		;		
		// State Change Condition
		IF (me.Alarm.eActivAlmClass<>E_AlmClass.EOFF) AND (me.Alarm.eActivAlmClass<>E_AlmClass.OFF) THEN	
			IF(me.intCmd=cBCC_CMD_READ) THEN
				me.StateMachine.intStateNext := cBCC_STA_READBusy;
			END_IF
		END_IF
	END_IF

//--------------------------------------------------------------------------------------
// Exit action
	IF (me.StateMachine.intState<>me.StateMachine.intStateNext) THEN
		;
	END_IF
END_METHOD

METHOD PROTECTED sta_OFFBusy : BOOL
// state implemetation
//--------------------------------------------------------------------------------------
// Entry action
	IF (me.StateMachine.intState<>me.StateMachine.intStateLastCycle) THEN
		me.StateMachine.intStateLastCycle := me.StateMachine.intState;
		
		// Simulation timer	
		fbSimulationTimer.IN := FALSE;
		fbSimulationTimer.PT := UDINT_TO_TIME(SIf.Par.udiTORead_ms / 2);
		fbSimulationTimer(); // set time/reset timer
		fbSimulationTimer.IN := TRUE; // start timer
		
	END_IF

//--------------------------------------------------------------------------------------
// Cyclic action
	IF (me.StateMachine.intState=me.StateMachine.intStateLastCycle) THEN
		
		// Simulation
		IF (CIf.SwCfg.bolSimulation) THEN
			fbSimulationTimer(); // simulation time
			IF (fbSimulationTimer.Q) THEN
				pBCD_SIf^.intCmd := cBCD_CMD_DONE;
			END_IF
		END_IF
			
		// State Change Condition
		IF (pBCD_SIf^.stErr.bolErrorActive = TRUE) THEN
			me.StateMachine.intStateNext :=  cSTA_ERROR;
		ELSIF(pBCD_SIf^.intCmd = cBCD_CMD_DONE) THEN
			me.StateMachine.intStateNext := cSTA_OFF;
		END_IF
	END_IF

//--------------------------------------------------------------------------------------
// Exit action
	IF (me.StateMachine.intState<>me.StateMachine.intStateNext) THEN
		;
	END_IF
END_METHOD

METHOD PROTECTED sta_PON : BOOL
// state implemetation
//--------------------------------------------------------------------------------------
// Entry action
	IF (me.StateMachine.intState<>me.StateMachine.intStateLastCycle) THEN
		me.StateMachine.intStateLastCycle := me.StateMachine.intState;
		
	END_IF


//--------------------------------------------------------------------------------------
// Cyclic action
	IF (me.StateMachine.intState=me.StateMachine.intStateLastCycle) THEN
		
		;	
		// State Change Condition
		IF (me.intCmd<>cCMD_PON) AND (me.intCmd<>cCMD_DONE) THEN
			me.StateMachine.intStateNext := cSTA_OFFBusy;
		END_IF
	END_IF


//--------------------------------------------------------------------------------------
// Exit action
	IF (me.StateMachine.intState<>me.StateMachine.intStateNext) THEN
		;
	END_IF
END_METHOD

METHOD PROTECTED sta_PONBusy : BOOL
// state implemetation
//--------------------------------------------------------------------------------------
// Entry action
	IF (me.StateMachine.intState<>me.StateMachine.intStateLastCycle) THEN
		me.StateMachine.intStateLastCycle := me.StateMachine.intState;
		
		// Simulation timer	
		fbSimulationTimer.IN := FALSE;
		fbSimulationTimer.PT := UDINT_TO_TIME(SIf.Par.udiTORead_ms / 2);
		fbSimulationTimer(); // set time/reset timer
		fbSimulationTimer.IN := TRUE; // start timer
		
		// Reset driver status
		pBCD_SIf^.stStatus.bolSocketConnected := FALSE;
		pBCD_SIf^.stStatus.bolComChecked := FALSE;
	END_IF

//--------------------------------------------------------------------------------------
// Cyclic action
	IF (me.StateMachine.intState=me.StateMachine.intStateLastCycle) THEN
			
		// Simulation
		IF (CIf.SwCfg.bolSimulation) THEN
			fbSimulationTimer(); // simulation time
			IF (fbSimulationTimer.Q) THEN
				// Set driver status
				pBCD_SIf^.stStatus.bolSocketConnected := TRUE;
				pBCD_SIf^.stStatus.bolComChecked := TRUE;		
			END_IF
		END_IF
			
		// Try to open the TCP socket		
		pBCD_SIf^.intCmd := cBCD_CMD_CONNECT_SOCKET;  
					
		// Check if socket connected
		IF (pBCD_SIf^.stStatus.bolSocketConnected = TRUE) THEN
			pBCD_SIf^.intCmd :=	cBCD_CMD_COM_TEST; // Execute a communication test to see if the device answer		
		END_IF
		
		// State Change Condition
		IF ((pBCD_SIf^.stErr.bolErrorActive = TRUE) OR (me.StateMachine.udiTimeInState_ms >= SIf.Par.udiTOPowerOn_ms)) THEN
			// SIf.Alm[2].strText := 'Initialisation error from barcode reader. No answer from device.';
			pfbAlarmCtrl^.setAlarm(CIf.Info.intCtrlId,2,0,ADR(SIf.Alm),E_AlmState.RST,CIf.Job.eMe_ActivAlmClass);
			me.StateMachine.intStateNext := cSTA_ERROR;				
		ELSIF (pBCD_SIf^.stStatus.bolComChecked = TRUE) THEN
			me.StateMachine.intStateNext := cSTA_PON;
		END_IF
	END_IF

//--------------------------------------------------------------------------------------
// Exit action
	IF (me.StateMachine.intState<>me.StateMachine.intStateNext) THEN
		;
	END_IF
END_METHOD

METHOD PROTECTED sta_READ : BOOL
// state implemetation
//--------------------------------------------------------------------------------------
// Entry action
	IF (me.StateMachine.intState<>me.StateMachine.intStateLastCycle) THEN
		me.StateMachine.intStateLastCycle := me.StateMachine.intState;

	END_IF

//--------------------------------------------------------------------------------------
// Cyclic action
	IF (me.StateMachine.intState=me.StateMachine.intStateLastCycle) THEN

		// Simulation
		IF (CIf.SwCfg.bolSimulation) THEN
			;
		END_IF
		
		// State Change Condition
		IF(me.intCmd=cBCC_CMD_READ) THEN
			me.StateMachine.intStateNext := cBCC_STA_READBusy;
		END_IF
	END_IF

//--------------------------------------------------------------------------------------
// Exit action
	IF (me.StateMachine.intState<>me.StateMachine.intStateNext) THEN
		;
	END_IF
END_METHOD

METHOD PROTECTED sta_READBusy : BOOL
// state implemetation
//--------------------------------------------------------------------------------------
// Entry action
	IF (me.StateMachine.intState<>me.StateMachine.intStateLastCycle) THEN
		me.StateMachine.intStateLastCycle := me.StateMachine.intState;
		
		// Simulation timer	
		fbSimulationTimer.IN := FALSE;
		fbSimulationTimer.PT := UDINT_TO_TIME(SIf.Par.udiTORead_ms / 2);
		fbSimulationTimer(); // set time/reset timer
		fbSimulationTimer.IN := TRUE; // start timer
		
		// Init
		SIf.Cur.bolNewCodeReaded:= FALSE;
		SIf.Cur.bolNoRead:= FALSE;
		SIf.Cur.stData.uliBarCode:= 0;
		SIf.Cur.stData.strBarCode:= '';
		
		// Read barcode
		pBCD_SIf^.intCmd := cBCD_CMD_READ_BARCODE;
	END_IF


//--------------------------------------------------------------------------------------
// Cyclic action
	IF (me.StateMachine.intState=me.StateMachine.intStateLastCycle) THEN

		// Simulation
		IF (CIf.SwCfg.bolSimulation) THEN
			fbSimulationTimer(); // simulation time
			IF (fbSimulationTimer.Q) THEN
				SIf.Cur.bolNewCodeReaded:= TRUE;
				uliSimBarCode:= uliSimBarCode + 1;
				pBCD_SIf^.stData.uliBarCode:= uliSimBarCode;
				pBCD_SIf^.stData.strBarCode:= ULINT_TO_STRING(pBCD_SIf^.stData.uliBarCode);
				pBCD_SIf^.intCmd := cBCD_CMD_DONE;		
			END_IF
		END_IF	

		// Check for new barcode
		IF (pBCD_SIf^.stData.uliBarCode <> uliBarCodeOld) AND (pBCD_SIf^.stData.uliBarCode<>0) THEN
			uliBarCodeOld:= pBCD_SIf^.stData.uliBarCode;
			SIf.Cur.bolNewCodeReaded:= TRUE;
		END_IF
		
		// Get data from driver
		SIf.Cur.stData.uliBarCode:= pBCD_SIf^.stData.uliBarCode;
		SIf.Cur.stData.strBarCode:= pBCD_SIf^.stData.strBarCode;			
		
		// State Change Condition
		IF (pBCD_SIf^.stErr.bolErrorActive = TRUE) THEN  
			me.StateMachine.intStateNext :=  cSTA_ERROR;
		ELSIF (me.StateMachine.udiTimeInState_ms > SIf.Par.udiTORead_ms) THEN
			// SIf.Alm[4].strText := 'Timeout wait on data';
			pfbAlarmCtrl^.setAlarm(CIf.Info.intCtrlId,4,0,ADR(SIf.Alm),E_AlmState.RST,CIf.Job.eMe_ActivAlmClass);
			me.StateMachine.intStateNext :=  cSTA_ERROR;
		ELSIF (pBCD_SIf^.intCmd = cBCD_CMD_DONE) THEN
			IF (SIf.Cur.stData.uliBarCode=0) THEN
				SIf.Cur.bolNoRead:= TRUE;
				uliBarCodeOld:= 0;
				// SIf.Alm[3].strText := 'Barcode could not be read. Answer *NoRead* from device';
				pfbAlarmCtrl^.setAlarm(CIf.Info.intCtrlId,3,0,ADR(SIf.Alm),E_AlmState.RST,CIf.Job.eMe_ActivAlmClass);	
			END_IF		
			me.StateMachine.intStateNext := cBCC_STA_READ;
		END_IF
	END_IF

//--------------------------------------------------------------------------------------
// Exit action
	IF (me.StateMachine.intState<>me.StateMachine.intStateNext) THEN
		CIf.Job.intACmd:= cCMD_DONE;
		CIf.Job.intMCmd:= cCMD_DONE;
	END_IF
END_METHOD

METHOD PROTECTED StateMachine : BOOL
SUPER^.StateMachine();

// main statemachine of base controller
CASE me.StateMachine.intState OF
    cBCC_STA_READBusy: 
        THIS^.sta_READBusy();
    cBCC_STA_READ: 
        THIS^.sta_READ();	
END_CASE;
END_METHOD

END_FUNCTION_BLOCK

// POUs/Controller/Lvl0/CYL (Cylinder)/FB_CYL
FUNCTION_BLOCK FB_CYL EXTENDS FB_CtrlBase

VAR_INPUT
	In_bolRetracted: BOOL;
	In_bolExtended: BOOL;
END_VAR
VAR_OUTPUT
	Out_bolRetract: BOOL;
	Out_bolExtend: BOOL;
END_VAR

VAR
	/// Specific interface struct for public access
	SIf: T_Ctrl_SIf_CYL;
END_VAR

(*__________________________________________________________________________________________________
¦	
¦	Vistaprint Schweiz GmbH
¦	CH - 8401 Winterthur
¦
¦	www.vistaprint.ch - info@vistaprint.ch
¦___________________________________________________________________________________________________

Function desription:
Cylinder implementation. 


History:
Version		Date			Author		Comment
---------------------------------------------------------------------------------------------------
0.00.1		25.04.2013		AVME/KVO	Start history
0.00.2		03.07.2013		AVME/KVO	Always call Super.always, no change to off when switch to automatic
										alarm evt EOFF, OFF or cmd off detection in Always
0.00.3		05.11.2013		AVME/KVO	integrate in BaseElements library, 
										FB alarm pointer used, alarm definition over ENUM
___________________________________________________________________________________________________*)


IF (me.bolActivate) THEN // cyclic call enabled
	IF (CIf.Info.bolInitDone=FALSE) THEN // first cycle -> init
		CtrlInit();
		CIf.Info.bolInitDone := TRUE;
	ELSE
		CycleStartDuty();
	
		Always();
		
		StateMachine();
		
		CycleEndDuty();
	END_IF
END_IF;

METHOD PROTECTED Always : BOOL
IF (me.bolChangeBackToAUTO=TRUE) THEN // switch mode to automatic switch off controller
	//me.StateMachine.intStateNext := cSTA_OFFBusy;
	me.bolChangeBackToAUTO := FALSE; // for cylinder no change to off when switch to automatic!!
END_IF

SUPER^.Always();

// ----------------------------------------------------------------------------------
// cyclic actions outside of statemachine
IF (me.StateMachine.intState<>cSTA_SINGLE_ANSWER) THEN
	
	; // always error supervision
	
END_IF

// ----------------------------------------------------------------------------------
// overrule error always from base -> no EOFF State!! in EOFF go to OFF
IF (me.StateMachine.intStateNext = cSTA_EOFFBusy) THEN
	IF (me.StateMachine.intState=cSTA_OFF) THEN
		me.StateMachine.intStateNext := cSTA_OFF;
	ELSE // stay in OFF
		me.StateMachine.intStateNext := cSTA_OFFBusy;
	END_IF
END_IF
END_METHOD

METHOD FB_init : BOOL
VAR_INPUT
	///if TRUE, the retain variables are initialized (warm start / cold start)
	bInitRetains: BOOL;
	///if TRUE, the instance afterwards gets moved into the copy code (online change)
	bInCopyCode: BOOL;
END_VAR
VAR
	ii: UINT;
END_VAR
//------------------------------------------------------------------------------------------------------------------------
// to manually change in new FUB implementation!!!
// define valid commands for this controller
FOR ii:= 0 TO (SIZEOF(CIf.Job.aCmdList)/SIZEOF(CIf.Job.aCmdList[0])-1) BY 1 DO
	IF (CIf.Job.aCmdList[ii].intCmd=cCMD_INITIALIZED) THEN
		// found first empty array element
		EXIT;
	END_IF
END_FOR

CIf.Job.aCmdList[ii].intCmd := cCMD_STOP;
CIf.Job.aCmdList[ii].strName := 'Stop'; 
CIf.Job.aCmdList[ii].bolAvailable := TRUE;
ii := ii +1;
CIf.Job.aCmdList[ii].intCmd := cCMD_RETRACT;
CIf.Job.aCmdList[ii].strName := 'Retract';
CIf.Job.aCmdList[ii].bolAvailable := TRUE;
ii := ii +1;
CIf.Job.aCmdList[ii].intCmd := cCMD_EXTEND; // for test simulation single answer
CIf.Job.aCmdList[ii].strName := 'Extend';
CIf.Job.aCmdList[ii].bolAvailable := TRUE;

// set name of class/typ
CIf.Info.strType := 'FB_CYL'; 

// set alarm class
SIf.Alm[E_ALM_CYL.SensorRetractAlwaysOn].eAlmClass := E_AlmClass.TSTOP;
SIf.Alm[E_ALM_CYL.SensorRetractAlwaysOn].strText := 'sensor retract always on'; 
SIf.Alm[E_ALM_CYL.SensorExtendNotReached].eAlmClass := E_AlmClass.TSTOP;
SIf.Alm[E_ALM_CYL.SensorExtendNotReached].strText := 'timeout extend - sensor extend not reached';
SIf.Alm[E_ALM_CYL.SensorExtendAlwaysOn].eAlmClass := E_AlmClass.TSTOP;
SIf.Alm[E_ALM_CYL.SensorExtendAlwaysOn].strText := 'sensor extend always on';
SIf.Alm[E_ALM_CYL.SensorRetractNotReached].eAlmClass := E_AlmClass.TSTOP;
SIf.Alm[E_ALM_CYL.SensorRetractNotReached].strText := 'timeout retract - sensor retract not reached';
SIf.Alm[E_ALM_CYL.InterlockExtend].eAlmClass := E_AlmClass.OFF;
SIf.Alm[E_ALM_CYL.InterlockExtend].strText := 'interlock extend - movement stopped';
SIf.Alm[E_ALM_CYL.InterlockRetract].eAlmClass := E_AlmClass.OFF;
SIf.Alm[E_ALM_CYL.InterlockRetract].strText := 'interlock retract - movement stopped';

//*******************************************************************************
// initial values
//*******************************************************************************

// Configuration defaults of class
CIf.SwCfg.bolExist := TRUE;
CIf.SwCfg.bolEnable := TRUE;
CIf.SwCfg.bolSimulation := FALSE;

// Parameter defaults of class
SIf.Par.udiExtendTime_ms := 10000;
SIf.Par.udiRetractTime_ms := 8000;
SIf.Par.udiSimExtendTime_ms := SIf.Par.udiExtendTime_ms/2;	
SIf.Par.udiSimRetractTime_ms := SIf.Par.udiRetractTime_ms/2;
END_METHOD

METHOD PROTECTED getCmdState : STRING
VAR_INPUT
	intCmdState: INT;
	bolState: BOOL;
END_VAR
getCmdState := SUPER^.getCmdState(intCmdState:=intCmdState,bolState:=bolState); // get global/base defined cmds/states
IF (getCmdState='') THEN // global not defined get local
	// get string cmd/state string information in runtime
	IF (bolState=FALSE) THEN
		// cmd's
		CASE intCmdState OF
			CYL_CmdState.cCMD_RETRACT: 
				getCmdState := 'cCMD_RETRACT';
			CYL_CmdState.cCMD_EXTEND: 
				getCmdState := 'cCMD_EXTEND';
		ELSE
			getCmdState := 'Cmd not defined';
		END_CASE;
	ELSE
	
	// cmd's
		CASE intCmdState OF
			CYL_CmdState.cSTA_RETRACTBusy: 
				getCmdState := 'cSTA_RETRACTBusy';
			CYL_CmdState.cSTA_RETRACT: 
				getCmdState := 'cSTA_RETRACT';
			CYL_CmdState.cSTA_EXTENDBusy: 
				getCmdState := 'cSTA_EXTENDBusy';
			CYL_CmdState.cSTA_EXTEND: 
				getCmdState := 'cSTA_EXTEND';
		ELSE
			getCmdState := 'State not defined';
		END_CASE;
	END_IF
END_IF
END_METHOD

METHOD getCtrlSIf : POINTER TO T_Ctrl_SIf_CYL
getCtrlSIf := ADR(SIf);
END_METHOD

METHOD PROTECTED IoInBridge : BOOL
// digitale and analoge inputs read from hardware or forcing
SIf.In.bolExtended.map := THIS^.In_bolExtended;
SIf.In.bolRetracted.map := THIS^.In_bolRetracted;

IF (CIf.SwCfg.bolSimulation = FALSE) THEN
	getInBol(CIf.Job.bolIoForce,ADR(SIf.In.bolExtended));
	getInBol(CIf.Job.bolIoForce,ADR(SIf.In.bolRetracted));
ELSE
	//simulation of global IO
END_IF
END_METHOD

METHOD PROTECTED IoOutBridge : BOOL
VAR
	bolSwitchValvesOff: BOOL;
END_VAR
// digitale and analoge inputs read from hardware or forcing
IF (CIf.SwCfg.bolSimulation = FALSE) THEN
	setOutBol(CIf.Job.bolIoForce ,ADR(SIf.Out.bolExtend));
	setOutBol(CIf.Job.bolIoForce ,ADR(SIf.Out.bolRetract));
	
	// check interlocks to prevent damages
	IF (CIf.Job.bolIlkOverwrite=FALSE) THEN
		bolSwitchValvesOff := FALSE;
		
		IF (SIf.Ilk.bolExtend=TRUE) THEN
			// switch off?
			IF (SIf.Cfg.eTyp = E_Typ_CYL.Valve1_Sensor0) OR (SIf.Cfg.eTyp = E_Typ_CYL.Valve1_Sensor2) 
				OR (SIf.Cfg.eTyp = E_Typ_CYL.Valve1_SensorExtended) OR (SIf.Cfg.eTyp = E_Typ_CYL.Valve1_SensorRetracted) THEN
				// monostabil valve -> do nothing
			ELSE
				// bistable valve ->  switch both off
				bolSwitchValvesOff := TRUE;
				IF (SIf.Out.bolExtend.map=1) THEN
					pfbAlarmCtrl^.setAlarm(CIf.Info.intCtrlId,E_ALM_CYL.InterlockExtend,0,ADR(SIf.Alm),E_AlmState.RST,CIf.Job.eMe_ActivAlmClass);
				END_IF
			END_IF
		END_IF
		
		IF (SIf.Ilk.bolRetract=TRUE) THEN
			// switch off?
			IF (SIf.Cfg.eTyp = E_Typ_CYL.Valve1_Sensor0) OR (SIf.Cfg.eTyp = E_Typ_CYL.Valve1_Sensor2) 
				OR (SIf.Cfg.eTyp = E_Typ_CYL.Valve1_SensorExtended) OR (SIf.Cfg.eTyp = E_Typ_CYL.Valve1_SensorRetracted) THEN
				// monostabil valve -> do nothing
				;
			ELSE
				// bistable valve -> switch both off
				bolSwitchValvesOff := TRUE;
				IF (SIf.Out.bolRetract.map=1) THEN
					pfbAlarmCtrl^.setAlarm(CIf.Info.intCtrlId,E_ALM_CYL.InterlockRetract,0,ADR(SIf.Alm),E_AlmState.RST,CIf.Job.eMe_ActivAlmClass);
				END_IF;
			END_IF
		END_IF
		
		// bistable valve -> switch both off
		IF (bolSwitchValvesOff) THEN
			SIf.Out.bolExtend.map := FALSE;
			SIf.Out.bolRetract.map := FALSE;
		END_IF
		
	END_IF

	THIS^.Out_bolExtend := SIf.Out.bolExtend.map;
	THIS^.Out_bolRetract := SIf.Out.bolRetract.map;
END_IF
END_METHOD

METHOD PROTECTED sta_ERROR : BOOL
// state implemetation
//--------------------------------------------------------------------------------------
// Entry action
	IF (me.StateMachine.intState<>me.StateMachine.intStateLastCycle) THEN
		me.StateMachine.intStateHistory := me.StateMachine.intStateLastCycle; // -> possibillity to go back to state before error
		me.StateMachine.intStateLastCycle := me.StateMachine.intState;
		
	END_IF


//--------------------------------------------------------------------------------------
// Cyclic action
	IF (me.StateMachine.intState=me.StateMachine.intStateLastCycle) THEN
		
		;
		
		
		// State Change Condition
		IF (CIf.Job.bolAlmReset = TRUE) THEN
			me.StateMachine.intStateNext := cSTA_ERRORQuit;
		END_IF
	END_IF




//--------------------------------------------------------------------------------------
// Exit action
	IF (me.StateMachine.intState<>me.StateMachine.intStateNext) THEN
		;
	END_IF
END_METHOD

METHOD PROTECTED sta_ERRORQuit : BOOL
// state implemetation
//--------------------------------------------------------------------------------------
// Entry action
	IF (me.StateMachine.intState<>me.StateMachine.intStateLastCycle) THEN
		me.StateMachine.intStateLastCycle := me.StateMachine.intState;
		
	END_IF


//--------------------------------------------------------------------------------------
// Cyclic action
	IF (me.StateMachine.intState=me.StateMachine.intStateLastCycle) THEN
		
		;
		// evtl. wait time if reset of device is necessary and then decide to go to states or ERROR state
		IF (CIf.Job.bolAlmReset = TRUE) THEN
			CIf.Job.eMe_ActivAlmClass := E_AlmClass.NONE; // reset feedback channel for parent
			CIf.Job.bolAlmReset := FALSE;
		END_IF
		
		// State Change Condition
		IF (CIf.Job.bolAlmReset = FALSE) THEN
			IF (me.StateMachine.intStateHistory<=cSTA_PON) THEN
				me.StateMachine.intStateNext := cSTA_PONBusy;
			ELSIF(me.intCmd=cCMD_OFF) THEN
				me.StateMachine.intStateNext := cSTA_OFFBusy;
			ELSIF(me.intCmd=cCMD_STOP) THEN
				me.StateMachine.intStateNext := cSTA_STOPBusy;
			ELSIF(me.intCmd=cCMD_RETRACT) THEN
				me.StateMachine.intStateNext := cSTA_RETRACTBusy;
			ELSIF(me.intCmd=cCMD_EXTEND) THEN
				me.StateMachine.intStateNext := cSTA_EXTENDBusy;
			END_IF
		END_IF
	END_IF


//--------------------------------------------------------------------------------------
// Exit action
	IF (me.StateMachine.intState<>me.StateMachine.intStateNext) THEN
		;
	END_IF
END_METHOD

METHOD PROTECTED sta_EXTEND : BOOL
// state implemetation
//--------------------------------------------------------------------------------------
// Entry action
	IF (me.StateMachine.intState<>me.StateMachine.intStateLastCycle) THEN
		me.StateMachine.intStateLastCycle := me.StateMachine.intState;

	END_IF


//--------------------------------------------------------------------------------------
// Cyclic action
	IF (me.StateMachine.intState=me.StateMachine.intStateLastCycle) THEN

		// Simulation
		IF (CIf.SwCfg.bolSimulation) THEN
			;
		END_IF
		
		// State Change Condition
		IF (SIf.In.bolRetracted.intern) THEN
			// sensor retract always on
			pfbAlarmCtrl^.setAlarm(CIf.Info.intCtrlId,E_ALM_CYL.SensorRetractAlwaysOn,0,ADR(SIf.Alm),E_AlmState.RST,CIf.Job.eMe_ActivAlmClass);
			me.StateMachine.intStateNext :=  cSTA_ERROR;
		ELSIF ((SIf.In.bolExtended.intern = FALSE) AND ((SIf.Cfg.eTyp = E_Typ_CYL.Valve1_SensorExtended) OR (SIf.Cfg.eTyp = E_Typ_CYL.Valve2_SensorExtended))) THEN // wait time until error?
			me.StateMachine.intStateNext := CYL_CmdState.cSTA_EXTENDBusy;
		ELSIF(me.intCmd=cCMD_STOP) THEN
			me.StateMachine.intStateNext := cSTA_STOPBusy;
		ELSIF(me.intCmd=CYL_CmdState.cCMD_RETRACT) THEN
			me.StateMachine.intStateNext := CYL_CmdState.cSTA_RETRACTBusy;
		END_IF
	END_IF



//--------------------------------------------------------------------------------------
// Exit action
	IF (me.StateMachine.intState<>me.StateMachine.intStateNext) THEN
		;
	END_IF
END_METHOD

METHOD PROTECTED sta_EXTENDBusy : BOOL
// state implemetation
//--------------------------------------------------------------------------------------
// Entry action
	IF (me.StateMachine.intState<>me.StateMachine.intStateLastCycle) THEN
		me.StateMachine.intStateLastCycle := me.StateMachine.intState;

		fbSimulationTimer.IN := FALSE;
		fbSimulationTimer.PT := UDINT_TO_TIME(SIf.Par.udiSimExtendTime_ms);
		fbSimulationTimer(); // set time/reset timer
		fbSimulationTimer.IN := TRUE; // start timer
	END_IF


//--------------------------------------------------------------------------------------
// Cyclic action
	IF (me.StateMachine.intState=me.StateMachine.intStateLastCycle) THEN

		// Simulation
		IF (CIf.SwCfg.bolSimulation) THEN
			fbSimulationTimer(); // simulation time
			IF (fbSimulationTimer.Q) THEN
				SIf.In.bolExtended.intern := TRUE;
				SIf.In.bolRetracted.intern := FALSE;
			END_IF
		END_IF
		
		//no change action
		SIf.Out.bolExtend.intern := TRUE;
		SIf.Out.bolRetract.intern := FALSE;
		
		
		// State Change Condition
		IF (me.StateMachine.udiTimeInState_ms>SIf.Par.udiExtendTime_ms) THEN
			IF (SIf.In.bolRetracted.intern) THEN
				// sensor retract always on
				pfbAlarmCtrl^.setAlarm(CIf.Info.intCtrlId,E_ALM_CYL.SensorRetractAlwaysOn,0,ADR(SIf.Alm),E_AlmState.RST,CIf.Job.eMe_ActivAlmClass);
			ELSE
				// timeout extend
				pfbAlarmCtrl^.setAlarm(CIf.Info.intCtrlId,E_ALM_CYL.SensorExtendNotReached,0,ADR(SIf.Alm),E_AlmState.RST,CIf.Job.eMe_ActivAlmClass);
			END_IF
			me.StateMachine.intStateNext :=  cSTA_ERROR;
		ELSIF (SIf.In.bolExtended.intern) AND (SIf.In.bolRetracted.intern=FALSE) THEN
			me.StateMachine.intStateNext := CYL_CmdState.cSTA_EXTEND;
		ELSIF ((SIf.Cfg.eTyp = E_Typ_CYL.Valve1_SensorRetracted) OR (SIf.Cfg.eTyp = E_Typ_CYL.Valve2_SensorRetracted))
				 AND (SIf.In.bolRetracted.intern=FALSE) AND (me.StateMachine.udiTimeInState_ms>SIf.Par.udiSimExtendTime_ms) THEN
			me.StateMachine.intStateNext := CYL_CmdState.cSTA_EXTEND;
		ELSIF ((SIf.Cfg.eTyp = E_Typ_CYL.Valve1_Sensor0) OR (SIf.Cfg.eTyp = E_Typ_CYL.Valve2_Sensor0))
				AND (me.StateMachine.udiTimeInState_ms>SIf.Par.udiSimExtendTime_ms) THEN
			me.StateMachine.intStateNext := CYL_CmdState.cSTA_EXTEND;		
		ELSIF(me.intCmd=cCMD_STOP) THEN
			me.StateMachine.intStateNext := cSTA_STOPBusy;
		ELSIF(me.intCmd=cCMD_RETRACT) THEN
			me.StateMachine.intStateNext := CYL_CmdState.cSTA_RETRACTBusy;
		END_IF
	END_IF




//--------------------------------------------------------------------------------------
// Exit action
	IF (me.StateMachine.intState<>me.StateMachine.intStateNext) THEN
		SIf.Cur.udiMoveTimeExtend := me.StateMachine.udiTimeInState_ms;
	END_IF
END_METHOD

METHOD PROTECTED sta_OFF : BOOL
// state implemetation
//--------------------------------------------------------------------------------------
// Entry action
	IF (me.StateMachine.intState<>me.StateMachine.intStateLastCycle) THEN
		me.StateMachine.intStateLastCycle := me.StateMachine.intState;
		
	END_IF


//--------------------------------------------------------------------------------------
// Cyclic action
	IF (me.StateMachine.intState=me.StateMachine.intStateLastCycle) THEN
		
		;
		
		// State Change Condition
		IF (me.Alarm.eActivAlmClass<>E_AlmClass.EOFF) AND (me.Alarm.eActivAlmClass<>E_AlmClass.OFF) THEN
			IF (me.intCmd=cCMD_STOP) THEN
				// sensor retract always on cylinder
				me.StateMachine.intStateNext :=  cSTA_STOPBusy;
			ELSIF (me.intCmd=CYL_CmdState.cCMD_EXTEND) THEN 
				me.StateMachine.intStateNext := cSTA_EXTENDBusy;
			ELSIF(me.intCmd=CYL_CmdState.cCMD_RETRACT) THEN
				me.StateMachine.intStateNext := cSTA_RETRACTBusy;
			END_IF
		END_IF
	END_IF




//--------------------------------------------------------------------------------------
// Exit action
	IF (me.StateMachine.intState<>me.StateMachine.intStateNext) THEN
		;
	END_IF
END_METHOD

METHOD PROTECTED sta_OFFBusy : BOOL
// state implemetation
//--------------------------------------------------------------------------------------
// Entry action
	IF (me.StateMachine.intState<>me.StateMachine.intStateLastCycle) THEN
		me.StateMachine.intStateLastCycle := me.StateMachine.intState;
		
	END_IF


//--------------------------------------------------------------------------------------
// Cyclic action
	IF (me.StateMachine.intState=me.StateMachine.intStateLastCycle) THEN
		
		// switch off?
		IF (SIf.Cfg.eTyp = E_Typ_CYL.Valve1_Sensor0) OR (SIf.Cfg.eTyp = E_Typ_CYL.Valve1_Sensor2) 
			OR (SIf.Cfg.eTyp = E_Typ_CYL.Valve1_SensorExtended) OR (SIf.Cfg.eTyp = E_Typ_CYL.Valve1_SensorRetracted) THEN
			// monostabil valve -> do nothing
			;
		ELSE
			// bistable valve -> switch both off
			SIf.Out.bolExtend.intern := FALSE;
			SIf.Out.bolRetract.intern := FALSE;
		END_IF
		
		
		
		// State Change Condition
		IF (TRUE) THEN
			me.StateMachine.intStateNext := cSTA_OFF;
		END_IF
	END_IF




//--------------------------------------------------------------------------------------
// Exit action
	IF (me.StateMachine.intState<>me.StateMachine.intStateNext) THEN
		;
	END_IF
END_METHOD

METHOD PROTECTED sta_PON : BOOL
// state implemetation
//--------------------------------------------------------------------------------------
// Entry action
	IF (me.StateMachine.intState<>me.StateMachine.intStateLastCycle) THEN
		me.StateMachine.intStateLastCycle := me.StateMachine.intState;
		
	END_IF


//--------------------------------------------------------------------------------------
// Cyclic action
	IF (me.StateMachine.intState=me.StateMachine.intStateLastCycle) THEN
		
		;
		
		// State Change Condition
		IF(me.intCmd=cCMD_STOP) THEN
			me.StateMachine.intStateNext := cSTA_STOPBusy;
		ELSIF(me.intCmd=cCMD_RETRACT) THEN
			me.StateMachine.intStateNext := cSTA_RETRACTBusy;
		ELSIF (me.intCmd=cCMD_EXTEND) THEN
			me.StateMachine.intStateNext := cSTA_EXTENDBusy;
		END_IF
	END_IF




//--------------------------------------------------------------------------------------
// Exit action
	IF (me.StateMachine.intState<>me.StateMachine.intStateNext) THEN
		;
	END_IF
END_METHOD

METHOD PROTECTED sta_RETRACT : BOOL
// state implemetation
//--------------------------------------------------------------------------------------
// Entry action
	IF (me.StateMachine.intState<>me.StateMachine.intStateLastCycle) THEN
		me.StateMachine.intStateLastCycle := me.StateMachine.intState;

	END_IF


//--------------------------------------------------------------------------------------
// Cyclic action
	IF (me.StateMachine.intState=me.StateMachine.intStateLastCycle) THEN

		// Simulation
		IF (CIf.SwCfg.bolSimulation) THEN
			;
		END_IF
		
		// State Change Condition
		IF (SIf.In.bolExtended.intern) THEN
			// sensor retract always on
			pfbAlarmCtrl^.setAlarm(CIf.Info.intCtrlId,E_ALM_CYL.SensorExtendAlwaysOn,0,ADR(SIf.Alm),E_AlmState.RST,CIf.Job.eMe_ActivAlmClass);
			me.StateMachine.intStateNext :=  cSTA_ERROR;
		ELSIF ((SIf.In.bolRetracted.intern = FALSE) AND ((SIf.Cfg.eTyp = E_Typ_CYL.Valve1_SensorRetracted) OR (SIf.Cfg.eTyp = E_Typ_CYL.Valve2_SensorRetracted))) THEN // wait time until error?
			me.StateMachine.intStateNext := CYL_CmdState.cSTA_RETRACTBusy;
		ELSIF(me.intCmd=cCMD_STOP) THEN
			me.StateMachine.intStateNext := cSTA_STOPBusy;
		ELSIF(me.intCmd=CYL_CmdState.cCMD_EXTEND) THEN
			me.StateMachine.intStateNext := CYL_CmdState.cSTA_EXTENDBusy;
		END_IF
	END_IF




//--------------------------------------------------------------------------------------
// Exit action
	IF (me.StateMachine.intState<>me.StateMachine.intStateNext) THEN
		;
	END_IF
END_METHOD

METHOD PROTECTED sta_RETRACTBusy : BOOL
// state implemetation
//--------------------------------------------------------------------------------------
// Entry action
	IF (me.StateMachine.intState<>me.StateMachine.intStateLastCycle) THEN
		me.StateMachine.intStateLastCycle := me.StateMachine.intState;
		
		SIf.Out.bolExtend.intern := FALSE;
		SIf.Out.bolRetract.intern := TRUE;
		
		fbSimulationTimer.IN := FALSE;
		fbSimulationTimer.PT := UDINT_TO_TIME(SIf.Par.udiSimRetractTime_ms);
		fbSimulationTimer(); // set time/reset timer
		fbSimulationTimer.IN := TRUE; // start timer
	END_IF


//--------------------------------------------------------------------------------------
// Cyclic action
	IF (me.StateMachine.intState=me.StateMachine.intStateLastCycle) THEN

		// Simulation
		IF (CIf.SwCfg.bolSimulation) THEN
			fbSimulationTimer(); // simulation time
			IF (fbSimulationTimer.Q) THEN
				SIf.In.bolRetracted.intern := TRUE;
				SIf.In.bolExtended.intern := FALSE;
			END_IF
		END_IF
		
		// State Change Condition
		IF (me.StateMachine.udiTimeInState_ms>SIf.Par.udiRetractTime_ms) THEN
			IF (SIf.In.bolExtended.intern) THEN
				// sensor extend always on 
				pfbAlarmCtrl^.setAlarm(CIf.Info.intCtrlId,E_ALM_CYL.SensorExtendAlwaysOn,0,ADR(SIf.Alm),E_AlmState.RST,CIf.Job.eMe_ActivAlmClass);
			ELSE
				// timeout retract cylinder
				pfbAlarmCtrl^.setAlarm(CIf.Info.intCtrlId,E_ALM_CYL.SensorRetractNotReached,0,ADR(SIf.Alm),E_AlmState.RST,CIf.Job.eMe_ActivAlmClass);
			END_IF
			me.StateMachine.intStateNext :=  cSTA_ERROR;
		ELSIF (SIf.In.bolRetracted.intern) AND(SIf.In.bolExtended.intern=FALSE) THEN
			me.StateMachine.intStateNext := CYL_CmdState.cSTA_RETRACT;
		ELSIF ((SIf.Cfg.eTyp = E_Typ_CYL.Valve1_SensorExtended) OR (SIf.Cfg.eTyp = E_Typ_CYL.Valve2_SensorExtended))
				 AND (SIf.In.bolExtended.intern=FALSE) AND (me.StateMachine.udiTimeInState_ms>SIf.Par.udiSimRetractTime_ms) THEN
			me.StateMachine.intStateNext := CYL_CmdState.cSTA_RETRACT;
		ELSIF ((SIf.Cfg.eTyp = E_Typ_CYL.Valve1_Sensor0) OR (SIf.Cfg.eTyp = E_Typ_CYL.Valve2_Sensor0))
				AND (me.StateMachine.udiTimeInState_ms>SIf.Par.udiSimRetractTime_ms) THEN
			me.StateMachine.intStateNext := CYL_CmdState.cSTA_RETRACT;		
		ELSIF(me.intCmd=cCMD_STOP) THEN
			me.StateMachine.intStateNext := cSTA_STOPBusy;
		ELSIF(me.intCmd=CYL_CmdState.cCMD_EXTEND) THEN
			me.StateMachine.intStateNext := CYL_CmdState.cSTA_EXTENDBusy;
		END_IF
	END_IF




//--------------------------------------------------------------------------------------
// Exit action
	IF (me.StateMachine.intState<>me.StateMachine.intStateNext) THEN
		SIf.Cur.udiMoveTimeRetract := me.StateMachine.udiTimeInState_ms;
	END_IF
END_METHOD

METHOD PROTECTED sta_STOP : BOOL
// state implemetation
//--------------------------------------------------------------------------------------
// Entry action
	IF (me.StateMachine.intState<>me.StateMachine.intStateLastCycle) THEN
		me.StateMachine.intStateLastCycle := me.StateMachine.intState;
		
	END_IF


//--------------------------------------------------------------------------------------
// Cyclic action
	IF (me.StateMachine.intState=me.StateMachine.intStateLastCycle) THEN
		
		;
		
		
		// State Change Condition
		IF (me.intCmd=CYL_CmdState.cCMD_EXTEND) THEN 
			me.StateMachine.intStateNext := CYL_CmdState.cSTA_EXTENDBusy;
		ELSIF(me.intCmd=CYL_CmdState.cCMD_RETRACT) THEN
			me.StateMachine.intStateNext := CYL_CmdState.cSTA_RETRACTBusy;
		END_IF
	END_IF




//--------------------------------------------------------------------------------------
// Exit action
	IF (me.StateMachine.intState<>me.StateMachine.intStateNext) THEN
		;
	END_IF
END_METHOD

METHOD PROTECTED sta_STOPBusy : BOOL
// state implemetation
//--------------------------------------------------------------------------------------
// Entry action
	IF (me.StateMachine.intState<>me.StateMachine.intStateLastCycle) THEN
		me.StateMachine.intStateLastCycle := me.StateMachine.intState;
		
	END_IF


//--------------------------------------------------------------------------------------
// Cyclic action
	IF (me.StateMachine.intState=me.StateMachine.intStateLastCycle) THEN
		
		// switch off?
		IF (SIf.Cfg.eTyp = E_Typ_CYL.Valve1_Sensor0) OR (SIf.Cfg.eTyp = E_Typ_CYL.Valve1_Sensor2) 
			OR (SIf.Cfg.eTyp = E_Typ_CYL.Valve1_SensorExtended) OR (SIf.Cfg.eTyp = E_Typ_CYL.Valve1_SensorRetracted) THEN
			// monostabil valve -> do nothing
			;
		ELSE
			// bistable valve -> switch both on -> block at position
			SIf.Out.bolExtend.intern := TRUE;
			SIf.Out.bolRetract.intern := TRUE;
		END_IF
		
		
		
		// State Change Condition
		IF (TRUE) THEN
			me.StateMachine.intStateNext := cSTA_STOP;
		END_IF
	END_IF




//--------------------------------------------------------------------------------------
// Exit action
	IF (me.StateMachine.intState<>me.StateMachine.intStateNext) THEN
		;
	END_IF
END_METHOD

METHOD PROTECTED StateMachine : BOOL
SUPER^.StateMachine();

// main statemachine of base controller
CASE me.StateMachine.intState OF
    CYL_CmdState.cSTA_RETRACTBusy: 
        THIS^.sta_RETRACTBusy();
    CYL_CmdState.cSTA_RETRACT: 
        THIS^.sta_RETRACT();
    CYL_CmdState.cSTA_EXTENDBusy: 
        THIS^.sta_EXTENDBusy();
    CYL_CmdState.cSTA_EXTEND: 
        THIS^.sta_EXTEND();
	cSTA_STOPBusy: 
        THIS^.sta_STOPBusy();
    cSTA_STOP: 
        THIS^.sta_STOP();
END_CASE;
END_METHOD

END_FUNCTION_BLOCK

// POUs/Controller/Lvl0/DRV (Drive)/FB_DRV
FUNCTION_BLOCK FB_DRV EXTENDS FB_CtrlBase
VAR_INPUT
	In_bolOverload: BOOL;
	In_bolPulse: BOOL;
	In_a_bolBlockedSupvervis: ARRAY[1..cMAX_BLOCKED_SUP] OF BOOL;
END_VAR
VAR_OUTPUT
	Out_bolSpeed_1: BOOL;
	Out_bolSpeed_2: BOOL;
END_VAR
VAR
	/// Specific interface struct for public access
	SIf: T_Ctrl_SIf_DRV;
	bolPulseFlag: BOOL;
	udiPulseTimeoutTimer: UDINT;
	/// Timer for speed average calculation
	udiTimerSpeedCalc: UDINT;
	/// Shift register for average calculation of the speed
	aSpeedShift: ARRAY[0..4] OF DINT;
	/// Size of Speed Shift array for average calculation
	intSpeedShiftSize: INT;
	/// Varible for Speedcalculation
	dinSpeedCalc_um_s: DINT;
	/// Varible for Speedcalculation
	dinSpeedNew_um_s: DINT;
	/// Old Position for Speed calculation
	dinPosOld_um: DINT;
	/// Loop variable
	intI: INT;
	/// Blocked supervision
	/// Array with supervision distances
	a_dintPinDistance: ARRAY[1..cMAX_BLOCKED_SUP] OF DINT;
	a_bolREBlockedSupvervis: ARRAY[1..cMAX_BLOCKED_SUP] OF BOOL;
	/// Old Position for from last cycle
	dinPosOldCycle_um: DINT;
END_VAR
VAR CONSTANT
	/// Check speed every 250ms
	cSpeedCalcTime_ms: UDINT := 250;
END_VAR

(*__________________________________________________________________________________________________
¦	
¦	Vistaprint Schweiz GmbH
¦	CH - 8401 Winterthur
¦
¦	www.vistaprint.ch - info@vistaprint.ch
¦___________________________________________________________________________________________________

Function desription:
Drive element for all different Drive types, 
Configuration of the type and Speed Calculation


History:
Version		Date			Author		Comment
---------------------------------------------------------------------------------------------------
0.00.1		27.06.2013		VP/RE		Start history
0.00.2		28.08.2013		AVME/PRE	Implement speed calculation
0.00.3		19.09.2013		AVME/PRE	Implement new Base Concept
0.00.4		02.10.2013		VP/RE		Added pulse counter. Changed pulse distance to 28.4 mm as a default value. Changed driving distance to 305 mm.
0.00.5      10.10.2013		AVME/DSC    In_bolBufferFull deleted. Not needed in DRV controller. Handled by parent controller if necessary.
0.00.6      18.10.2013		AVME/DSC    SIf.Alm[4].strText deleted in FB_init. Not used anymore.
0.00.7		22.10.2013		AVME/MRU	DRV without pulse sensor simulated pulse imroved
0.00.8      23.10.2013		AVME/DSC    Speed calculation from always to state RUN. cSpeedCalcTime_ms -> 250ms. Shift register array 0..4. Clear buffer in state RUN entry action.
										Changes for better position interpolation in controllers like MER, DPJ, DHC and JUN.
___________________________________________________________________________________________________*)


IF (me.bolActivate) THEN // cyclic call enabled
	IF (CIf.Info.bolInitDone=FALSE) THEN // first cycle -> init
		CtrlInit();
		CIf.Info.bolInitDone := TRUE;
	ELSE
		CycleStartDuty();
	
		Always();
		
		StateMachine();
		
		CycleEndDuty();
	END_IF
END_IF;

METHOD PROTECTED Always : BOOL
SUPER^.Always();

IF (me.StateMachine.intState<>cSTA_SINGLE_ANSWER) THEN
	
	// Error checks not in OFF and Error States
	IF (me.StateMachine.intState<>cSTA_OFF) AND (me.StateMachine.intState<>cSTA_ERROR) AND (me.StateMachine.intState<>cSTA_ERRORQuit) THEN
		IF SIf.In.bolOverload.intern THEN
			// SIf.Alm[1].strText := 'Drive overload'; 
			pfbAlarmCtrl^.setAlarm(CIf.Info.intCtrlId,1,0,ADR(SIf.Alm),E_AlmState.RST,CIf.Job.eMe_ActivAlmClass);		
			me.StateMachine.intStateNext := cSTA_ERROR;		
		END_IF
		
		// Blocked Supervision control
		// Sensor detect Pins, if a defined count of pins are brocken, the machine stops
		FOR intI := 1 TO SIf.Cfg.usiCountBlockedSupervis DO
			
			// Simulation
			// Simulate the Pins in the drive
			IF (CIf.SwCfg.bolSimulation) THEN
				IF (a_dintPinDistance[intI] >  SIf.Cfg.dinPinDistance_um) THEN
					SIf.In.a_bolBlockedSupvervis[intI].intern := TRUE;
				ELSE
					SIf.In.a_bolBlockedSupvervis[intI].intern := FALSE;
				END_IF
			END_IF
		
			// Check if a new pin is arrive, set distance to last pin to '0'
			IF ((SIf.In.a_bolBlockedSupvervis[intI].intern = TRUE) AND (a_bolREBlockedSupvervis[intI] = FALSE)) THEN
				a_bolREBlockedSupvervis[intI] := TRUE;
				a_dintPinDistance[intI] := 0;
			ELSIF ((SIf.In.a_bolBlockedSupvervis[intI].intern = FALSE) AND (a_bolREBlockedSupvervis[intI] = TRUE)) THEN
				a_bolREBlockedSupvervis[intI] := FALSE;
			END_IF
			// Check distance to last Pin, if to far away, set error
			IF (a_dintPinDistance[intI] > ((SIf.Par.int_MaxBrokenPins+1) * SIf.Cfg.dinPinDistance_um)) THEN
				// SIf.Alm[3].strText := 'Drive blocked, Pins are broken'; 
				pfbAlarmCtrl^.setAlarm(CIf.Info.intCtrlId,3,0,ADR(SIf.Alm),E_AlmState.RST,CIf.Job.eMe_ActivAlmClass);
				a_dintPinDistance[intI] := 0;		
				me.StateMachine.intStateNext := cSTA_ERROR;		
			ELSE
				a_dintPinDistance[intI] := a_dintPinDistance[intI] + SIf.Cur.dinPos_um - dinPosOldCycle_um;					
			END_IF		
		END_FOR
		dinPosOldCycle_um := SIf.Cur.dinPos_um;
	END_IF
END_IF

// Speed calculation in always function to get correct position everytime, not only in run
// observe no pulse detected failure case 
IF (SIf.In.bolPulse.intern AND NOT(bolPulseFlag)) THEN				
	// calculate CUR
	SIf.Cur.dinPos_um := SIf.Cur.dinPos_um + SIf.Cfg.dinDistPerPulse_um;
	SIf.Cur.dinPulseCounter := SIf.Cur.dinPulseCounter + 1;
		
	udiPulseTimeoutTimer := 0;
	bolPulseFlag := TRUE;
ELSIF (NOT(SIf.In.bolPulse.intern) AND bolPulseFlag) THEN
	bolPulseFlag := FALSE;
END_IF

// Always change actions in Base Library
// ----------------------------------------------------------------------------------
// overrule error always from base -> no EOFF State!! in EOFF go to OFF
IF (me.StateMachine.intStateNext = cSTA_EOFFBusy) THEN
	IF (me.StateMachine.intState=cSTA_OFF) THEN
		me.StateMachine.intStateNext := cSTA_OFF;
	ELSE // stay in OFF
		me.StateMachine.intStateNext := cSTA_OFFBusy;
	END_IF
END_IF
END_METHOD

METHOD FB_init : BOOL
VAR_INPUT
	///if TRUE, the retain variables are initialized (warm start / cold start)
	bInitRetains: BOOL;
	///if TRUE, the instance afterwards gets moved into the copy code (online change)
	bInCopyCode: BOOL;
END_VAR
VAR
	ii: UINT;
END_VAR
//------------------------------------------------------------------------------------------------------------------------
// to manually change in new FUB implementation!!!
// define valid commands for this controller
FOR ii:= 0 TO (SIZEOF(CIf.Job.aCmdList)/SIZEOF(CIf.Job.aCmdList[0])-1) BY 1 DO
	IF (CIf.Job.aCmdList[ii].intCmd=cCMD_INITIALIZED) THEN
		// found first empty array element
		EXIT;
	END_IF
END_FOR
CIf.Job.aCmdList[ii].intCmd := cCMD_RUN;
CIf.Job.aCmdList[ii].strName := 'Run'; 
CIf.Job.aCmdList[ii].bolAvailable := TRUE;
ii := ii +1;

// set name of class/typ
CIf.Info.strType := 'FB_DRV'; 

// set alarm class
SIf.Alm[1].eAlmClass := E_AlmClass.OFF;
SIf.Alm[1].strText := 'Drive overload'; 
SIf.Alm[2].eAlmClass := E_AlmClass.OFF;
SIf.Alm[2].strText := 'Timeout no pulse detected';
SIf.Alm[3].eAlmClass := E_AlmClass.OFF;
SIf.Alm[3].strText := 'Drive blocked, Pins are broken'; 

//*******************************************************************************
// initial values
//*******************************************************************************

// software configuration
CIf.SwCfg.bolExist := TRUE;
CIf.SwCfg.bolSimulation := FALSE;

// parmeter
SIf.Par.udi_pulseTimeout_ms := 2000;
SIf.Par.udi_pulseSim_ms := 56;
SIf.Par.usi_speedLevel := 0;
SIf.Par.int_MaxBrokenPins := 5;

SIf.Cfg.dinDistPerPulse_um := 28400; // 28,4[mm/puls]
SIf.Cfg.usiCountBlockedSupervis := 0;
SIf.Cfg.dinPinDistance_um := 305000;
END_METHOD

METHOD getCtrlSIf : POINTER TO T_Ctrl_SIf_DRV
getCtrlSIf := ADR(SIf);
END_METHOD

METHOD PROTECTED IoInBridge : BOOL
// digitale and analoge inputs read from hardware or forcing
SIf.In.bolOverload.map := THIS^.In_bolOverload;
SIf.In.bolPulse.map := THIS^.In_bolPulse;

FOR intI := 1 TO SIf.Cfg.usiCountBlockedSupervis DO
	SIf.In.a_bolBlockedSupvervis[intI].map := THIS^.In_a_bolBlockedSupvervis[intI];
	IF (CIf.SwCfg.bolSimulation = FALSE) THEN
		getInBol(CIf.Job.bolIoForce,ADR(SIf.In.a_bolBlockedSupvervis[intI]));
	END_IF
END_FOR

IF (CIf.SwCfg.bolSimulation = FALSE) THEN
	getInBol(CIf.Job.bolIoForce,ADR(SIf.In.bolOverload));
	getInBol(CIf.Job.bolIoForce,ADR(SIf.In.bolPulse));
	//ctrl.In.bol_PosSwitchBasicDefTyp.intern := getInBol(ctrl.ifc.Job.bol_Force ,ADR(ctrl.In.bol_PosSwitchBasicDefTyp);
ELSE
	//simulation of global IO
	SIf.In.bolOverload.intern := FALSE;
END_IF
END_METHOD

METHOD PROTECTED IoOutBridge : BOOL
VAR
	bolSwitchValvesOff: BOOL;
END_VAR
// digitale and analoge inputs read from hardware or forcing
IF (CIf.SwCfg.bolSimulation = FALSE) THEN
	setOutBol(CIf.Job.bolIoForce ,ADR(SIf.Out.bolSpeed_1));
	setOutBol(CIf.Job.bolIoForce ,ADR(SIf.Out.bolSpeed_2));

	THIS^.Out_bolSpeed_1 := SIf.Out.bolSpeed_1.map;
	THIS^.Out_bolSpeed_2 := SIf.Out.bolSpeed_2.map;
END_IF
END_METHOD

METHOD PRIVATE SetSpeed
// 0=slow, 1=middle, 2=fast
CASE SIf.Par.usi_speedLevel OF
	0:
		SIf.Out.bolSpeed_1.intern := TRUE;
		SIf.Out.bolSpeed_2.intern := FALSE;
	1:
		SIf.Out.bolSpeed_1.intern := TRUE;
		SIf.Out.bolSpeed_2.intern := TRUE;
	2:
		SIf.Out.bolSpeed_1.intern := FALSE;
		SIf.Out.bolSpeed_2.intern := TRUE;
	ELSE
		SIf.Out.bolSpeed_1.intern := TRUE;
		SIf.Out.bolSpeed_2.intern := FALSE;
END_CASE
END_METHOD

METHOD PROTECTED sta_ERROR : BOOL
// state implemetation
//--------------------------------------------------------------------------------------
// Entry action
IF (me.StateMachine.intState<>me.StateMachine.intStateLastCycle) THEN
	me.StateMachine.intStateHistory := me.StateMachine.intStateLastCycle; // -> possibillity to go back to state before error
	me.StateMachine.intStateLastCycle := me.StateMachine.intState;
	
	SIf.Out.bolSpeed_1.intern := FALSE;
	SIf.Out.bolSpeed_2.intern := FALSE;
	
END_IF


//--------------------------------------------------------------------------------------
// Cyclic action
	IF (me.StateMachine.intState=me.StateMachine.intStateLastCycle) THEN
		
		;
		
		
		// State Change Condition
		IF (CIf.Job.bolAlmReset = TRUE) THEN
			me.StateMachine.intStateNext := cSTA_ERRORQuit;
		END_IF
	END_IF




//--------------------------------------------------------------------------------------
// Exit action
	IF (me.StateMachine.intState<>me.StateMachine.intStateNext) THEN
		;
	END_IF
END_METHOD

METHOD PROTECTED sta_OFF : BOOL
// state implemetation
//--------------------------------------------------------------------------------------
// Entry action
	IF (me.StateMachine.intState<>me.StateMachine.intStateLastCycle) THEN
		me.StateMachine.intStateLastCycle := me.StateMachine.intState;
		
	END_IF


//--------------------------------------------------------------------------------------
// Cyclic action
	IF (me.StateMachine.intState=me.StateMachine.intStateLastCycle) THEN
		
		;
		
		
		// State Change Condition
		IF (me.Alarm.eActivAlmClass<>E_AlmClass.EOFF) AND (me.Alarm.eActivAlmClass<>E_AlmClass.OFF) THEN
			IF (me.intCmd=cCMD_RUN) THEN 
				me.StateMachine.intStateNext := cSTA_RUNBusy;
			END_IF
		END_IF
	END_IF




//--------------------------------------------------------------------------------------
// Exit action
	IF (me.StateMachine.intState<>me.StateMachine.intStateNext) THEN
		;
	END_IF
END_METHOD

METHOD PROTECTED sta_OFFBusy : BOOL
// state implemetation
//--------------------------------------------------------------------------------------
// Entry action
	IF (me.StateMachine.intState<>me.StateMachine.intStateLastCycle) THEN
		me.StateMachine.intStateLastCycle := me.StateMachine.intState;
		
	END_IF


//--------------------------------------------------------------------------------------
// Cyclic action
	IF (me.StateMachine.intState=me.StateMachine.intStateLastCycle) THEN
		
		SIf.Out.bolSpeed_1.intern := FALSE;
		SIf.Out.bolSpeed_2.intern := FALSE;
		
		// State Change Condition
		IF (TRUE) THEN
			me.StateMachine.intStateNext := cSTA_OFF;
		END_IF
	END_IF




//--------------------------------------------------------------------------------------
// Exit action
	IF (me.StateMachine.intState<>me.StateMachine.intStateNext) THEN
		;
	END_IF
END_METHOD

METHOD PROTECTED sta_PON : BOOL
// state implemetation
//--------------------------------------------------------------------------------------
// Entry action
	IF (me.StateMachine.intState<>me.StateMachine.intStateLastCycle) THEN
		me.StateMachine.intStateLastCycle := me.StateMachine.intState;
		
	END_IF


//--------------------------------------------------------------------------------------
// Cyclic action
	IF (me.StateMachine.intState=me.StateMachine.intStateLastCycle) THEN
		
		;
		
		
		// State Change Condition
		IF ((me.intCmd=cCMD_OFF) OR (me.intCmd=cCMD_RUN)) THEN
			me.StateMachine.intStateNext := cSTA_OFFBusy;
		END_IF
	END_IF




//--------------------------------------------------------------------------------------
// Exit action
	IF (me.StateMachine.intState<>me.StateMachine.intStateNext) THEN
		;
	END_IF
END_METHOD

METHOD PROTECTED sta_RUN : BOOL
VAR
	ii: INT;
END_VAR
// state implemetation
//--------------------------------------------------------------------------------------
// Entry action
	IF (me.StateMachine.intState<>me.StateMachine.intStateLastCycle) THEN
		me.StateMachine.intStateLastCycle := me.StateMachine.intState;
		
		udiPulseTimeoutTimer := 0;
		bolPulseFlag := FALSE;
		
		fbSimulationTimer.IN := FALSE;
		fbSimulationTimer.PT := UDINT_TO_TIME(SIf.Par.udi_pulseSim_ms);  
		fbSimulationTimer(); // set time/reset timer
		fbSimulationTimer.IN := TRUE; // start timer
			
		// Get Size of array
		intSpeedShiftSize := SIZEOF(aSpeedShift)/(SIZEOF(aSpeedShift[0]));
		// Clear speed buffer
		FOR ii:=0 TO intSpeedShiftSize-1 BY 1 DO
			aSpeedShift[ii]:=0;
		END_FOR
		
	END_IF


//--------------------------------------------------------------------------------------
// Cyclic action
	IF (me.StateMachine.intState=me.StateMachine.intStateLastCycle) THEN
		
		// Simulation
		// AND speed simulation if no distance sensor is existing !!!
		IF ((CIf.SwCfg.bolSimulation) OR (SIf.Cfg.bolPulseExist = FALSE)) THEN
			fbSimulationTimer(); // simulation time
			IF (fbSimulationTimer.Q) THEN
				SIf.In.bolPulse.intern := TRUE; 
				In_bolPulse := TRUE; // MRU 22.10.2013 added for drive without pulse sensor
				fbSimulationTimer.IN := FALSE;
			ELSE
				SIf.In.bolPulse.intern := FALSE;
				In_bolPulse := FALSE; // MRU 22.10.2013 added for drive without pulse sensor
				fbSimulationTimer.IN := TRUE;
			END_IF
		END_IF
	
		IF SIf.Cfg.bolSpeedVariable = TRUE THEN
			SetSpeed();
		END_IF;
		
		udiPulseTimeoutTimer := udiPulseTimeoutTimer + me.FUBInfo.udiSample_ms;
		
		
		// Speed calculation
		IF udiTimerSpeedCalc >= cSpeedCalcTime_ms THEN
			dinSpeedNew_um_s := (SIf.Cur.dinPos_um - dinPosOld_um)*1000 / UDINT_TO_DINT(udiTimerSpeedCalc);
			dinSpeedCalc_um_s := dinSpeedNew_um_s;
			// Get Size of array
			intSpeedShiftSize := SIZEOF(aSpeedShift)/(SIZEOF(aSpeedShift[0]));
			intI := intSpeedShiftSize-1;
			WHILE intI > 0 DO		
				// Shift all speeds one field
				aSpeedShift[intI] := aSpeedShift[intI-1];
				dinSpeedCalc_um_s := dinSpeedCalc_um_s + aSpeedShift[intI];
				intI := intI - 1;
			END_WHILE
			aSpeedShift[0] := dinSpeedNew_um_s;
			SIf.Cur.dinSpeed_um_s := dinSpeedCalc_um_s / intSpeedShiftSize;
			dinPosOld_um := SIf.Cur.dinPos_um;
			udiTimerSpeedCalc := 0;
				
		ELSE
			udiTimerSpeedCalc := udiTimerSpeedCalc + me.FUBInfo.udiSample_ms;
		END_IF
		
		
		// State Change Condition
		IF ((udiPulseTimeoutTimer >= Sif.Par.udi_pulseTimeout_ms) AND (SIf.Cfg.bolPulseExist = TRUE)) THEN
			// SIf.Alm[2].strText := 'Timeout no pulse detected';
			pfbAlarmCtrl^.setAlarm(CIf.Info.intCtrlId,2,0,ADR(SIf.Alm),E_AlmState.RST,CIf.Job.eMe_ActivAlmClass);

			me.StateMachine.intStateNext :=  cSTA_ERROR;		
		ELSIF (me.intCmd=cCMD_OFF) THEN
			me.StateMachine.intStateNext :=  cSTA_OFFBusy;
		END_IF
		
	END_IF



//--------------------------------------------------------------------------------------
// Exit action
	IF (me.StateMachine.intState<>me.StateMachine.intStateNext) THEN
		// Set speed zero
		SIf.Cur.dinSpeed_um_s := 0;
	END_IF
END_METHOD

METHOD PROTECTED sta_RUNBusy : BOOL
// state implemetation
//--------------------------------------------------------------------------------------
// Entry action
	IF (me.StateMachine.intState<>me.StateMachine.intStateLastCycle) THEN
		me.StateMachine.intStateLastCycle := me.StateMachine.intState;
		
	END_IF


//--------------------------------------------------------------------------------------
// Cyclic action
	IF (me.StateMachine.intState=me.StateMachine.intStateLastCycle) THEN

		IF SIf.Cfg.bolSpeedVariable = TRUE THEN
			SetSpeed();
		ELSE
			SIf.Out.bolSpeed_1.intern := TRUE;
		END_IF;		
		
		// State Change Condition
		IF (TRUE) THEN
			me.StateMachine.intStateNext := cSTA_RUN;
		END_IF
	END_IF




//--------------------------------------------------------------------------------------
// Exit action
	IF (me.StateMachine.intState<>me.StateMachine.intStateNext) THEN
		;
	END_IF
END_METHOD

METHOD PROTECTED StateMachine : BOOL
SUPER^.StateMachine();

// main statemachine of base controller
CASE me.StateMachine.intState OF
    cSTA_RUNBusy: 
        THIS^.sta_RUNBusy();
    cSTA_RUN: 
        THIS^.sta_RUN();
END_CASE;
END_METHOD

END_FUNCTION_BLOCK

// POUs/Controller/Lvl0/RFW (RFID Reader-Writer)/FB_DtChnToLine_NewRFID
FUNCTION_BLOCK FB_DtChnToLine_NewRFID
VAR_INPUT
	bolResetError: BOOL;
	pSIf: POINTER TO T_Ctrl_SIf_RFW;
END_VAR
VAR_OUTPUT
	///Error value
	intError: INT;
END_VAR
VAR
	/// Internal Variable
	intStatemachine: INT;
	/// Time Variables
	fbGetSystemTime: GETSYSTEMTIME;
	stfileTime: T_FILETIME;
	dtActualTime: DT;
	/// Data not correct
	bolDataBad: BOOL;
	/// Retry Counts for error message
	intCountRetry: INT;
	/// Buffer for Senddata
	aBuffer: ARRAY[0..cDtChnBuffer] OF T_NewRFID_DtChn;
	/// Pointer for new Input
	intPBufferInput: INT;
	/// Pointer for readout
	intPBufferOutput: INT;
	/// Data Channel Specific Variable
	intIndexOldest: INT;
	/// Date and time of the oldes imput
	dtOldestTag: DT;
END_VAR
VAR CONSTANT
	cDtChnBuffer: INT := 20;
	cSTA_SUB_Data_Init: INT := 900;
	cSTA_SUB_Data_WaitForJob: INT := 902;
	cSTA_SUB_Data_SendData: INT := 904;
	cSTA_SUB_Data_Acknowledge: INT := 906;
	cSTA_SUB_Data_Retry: INT := 908;
	cSTA_SUB_Data_Error: INT := 910;
	cDataState_DONE: INT := -1;
	cDataState_Ready: INT := 1;
	cDataState_Retry: INT := -99;
	cDataState_Error: INT := -100;
	cMAX_RETRY: INT := 10;
	/// Error Codes
	cERR_BufferFull: INT := -99;
	cERR_NoSIF: INT := -100;
END_VAR

(*__________________________________________________________________________________________________
¦	
¦	Vistaprint Schweiz GmbH
¦	CH - 8401 Winterthur
¦
¦	www.vistaprint.ch - info@vistaprint.ch
¦___________________________________________________________________________________________________

Function desription:
Datachannel to send data to Lince Controller
Insert new Job with Method Creat in a Buffer
Send buffer elements if Linecontroller is ready


History:
Version		Date			Author		Comment
---------------------------------------------------------------------------------------------------
0.00.1		26.08.2013		AVM/PRE		Start history
0.00.2		30.09.2013		AVM/PRE		Date and time with string, not with DT Type

___________________________________________________________________________________________________*)

// Data Channel to Receive Data from Line Controller
// Startup check States
IF (pSIf <> 0) THEN
	IF (intStatemachine < cSTA_SUB_Data_Init) THEN
		intStatemachine := cSTA_SUB_Data_Init;
	END_IF
ELSE
	intError := cERR_NoSIF;
END_IF

CASE intStatemachine OF
	cSTA_SUB_Data_Init:
		IF pSIf^.DtChnToLine.stNewRfid.intDataState = cDataState_DONE THEN
			intStatemachine := cSTA_SUB_Data_WaitForJob;
		END_IF
		
	cSTA_SUB_Data_WaitForJob:
		// New data arrived
		IF intPBufferInput <> intPBufferOutput THEN
			IF pSIf^.DtChnToLine.stNewRfid.intDataState = cDataState_DONE THEN
				intStatemachine := cSTA_SUB_Data_SendData;
			END_IF
		END_IF
	
	cSTA_SUB_Data_SendData:	
		pSIf^.DtChnToLine.stNewRfid.uliTagID := aBuffer[intPBufferOutput].uliTagID;
		pSIf^.DtChnToLine.stNewRfid.strID := aBuffer[intPBufferOutput].strID;
		pSIf^.DtChnToLine.stNewRfid.strTimestamp := aBuffer[intPBufferOutput].strTimestamp;
		pSIf^.DtChnToLine.stNewRfid.intDataState := cDataState_Ready;
		intStatemachine := cSTA_SUB_Data_Acknowledge;	
		
	cSTA_SUB_Data_Acknowledge:	
		IF pSIf^.DtChnToLine.stNewRfid.intDataState = cDataState_DONE THEN
			// Data read from Line Controller
			// Reset Buffer Element
			aBuffer[intPBufferOutput].strTimestamp := '';
			aBuffer[intPBufferOutput].intDataState := 0;
			aBuffer[intPBufferOutput].uliTagID := 0;
			aBuffer[intPBufferOutput].strID := '';
			// Increase Read out pointer
			IF intPBufferOutput < cDtChnBuffer THEN
				intPBufferOutput := intPBufferOutput + 1;
			ELSE
				intPBufferOutput := 0;
			END_IF
			intStatemachine := cSTA_SUB_Data_WaitForJob;
			
		ELSIF pSIf^.DtChnToLine.stNewRfid.intDataState = cDataState_Retry THEN
			intStatemachine := cSTA_SUB_Data_Retry;
		ELSIF pSIf^.DtChnToLine.stNewRfid.intDataState = cDataState_Error THEN
			intStatemachine := cSTA_SUB_Data_Error;
		END_IF
		
	cSTA_SUB_Data_Retry:
			IF intCountRetry < cMAX_RETRY THEN
				intCountRetry := intCountRetry + 1;
				intStatemachine := cSTA_SUB_Data_SendData;
			ELSE
				intStatemachine := cSTA_SUB_Data_Error;
			END_IF

	cSTA_SUB_Data_Error:
		intError := intCountRetry;
		IF bolResetError = TRUE THEN
			intStatemachine := cSTA_SUB_Data_WaitForJob;
		END_IF
			
END_CASE

METHOD Creat : INT
VAR_INPUT
	/// configurable if Tag or Tray ID
	In_strID: STRING;
	In_uliTagID: ULINT;
END_VAR

VAR
	strTemp : STRING;
END_VAR
// Insert a new Job to send at Line controller
// Only insert the job, if the buffer is not full, next input dosn't cross input and Outputpointer

// Get Systemtime
fbGetSystemTime(timeLoDW=>stfileTime.dwLowDateTime, timeHiDW=>stfileTime.dwHighDateTime);
dtActualTime := FILETIME_TO_DT( stfileTime );

IF ((intPBufferInput + 1) = intPBufferOutput) OR ((intPBufferInput = cDtChnBuffer) AND (intPBufferOutput = 0)) THEN
	Creat := cERR_BufferFull;
ELSE
	aBuffer[intPBufferInput].uliTagID := In_uliTagID;
	aBuffer[intPBufferInput].strID := In_strID;
	strTemp := DT_TO_STRING(dtActualTime);
	strTemp := Tc2_Standard.RIGHT(STR:=strTemp, SIZE:= (LEN(strTemp)-3));
	strTemp := CONCAT(strTemp,'.000');	
	aBuffer[intPBufferInput].strTimestamp := strTemp;
	IF intPBufferInput < cDtChnBuffer THEN
		intPBufferInput := intPBufferInput + 1;
	ELSE
		intPBufferInput := 0;
	END_IF
	Creat := intPBufferInput;
END_IF
END_METHOD

END_FUNCTION_BLOCK

// POUs/Controller/Lvl0/RFW (RFID Reader-Writer)/FB_RFW
FUNCTION_BLOCK FB_RFW EXTENDS FB_CtrlBase
VAR_INPUT
	pRFD_SIf: POINTER TO T_RFD;
END_VAR
VAR
	/// Specific interface struct for public access
	SIf: T_Ctrl_SIf_RFW;
	/// Internal Variable
	bolNewTag: BOOL;
	/// Rising Edge New tag at antenna
	bolRENewTag: BOOL;
	/// Read All is finished
	bolAllFinished: BOOL;
	/// Internal Job for more reading
	dwoJobIntern: DWORD;
	/// Startadress on the Tag from the needed Data
	uinDataAdress: UINT;
	/// Lengh of data to read or write
	uinDataLengh: UINT;
	/// old Tag ID to know a new RFID Tag is on antenna
	uliTagID_old: ULINT;
	/// Temporary Help Variable
	usiTemp: USINT;
	/// Temporary Help Variable
	uinTemp: UINT;
	/// Temporary Help Variable
	intTemp: INT;
	intValue: INT;
	/// Temporary Help Variable
	udiTemp: UDINT;
	/// Temporary Help Variable
	uliTemp: LWORD;
	/// Temporary Help Variable
	strTemp: STRING;
	/// Temporary Help Variable to save to position of the point in the string
	intPositionPoint: INT;
	/// Temporary Help Variable to save to position of the - in the string
	intPositionSign: INT;
	/// Short Brake between the different Reads
	udiTimeDelayRead : UDINT;
	/// Data Channel to Line new RFID Tag
	fbDtChnToLine_NewRFID: FB_DtChnToLine_NewRFID;
	intDtChnToLineState: INT;

END_VAR
VAR CONSTANT
	///sub States for RUN Function
	cRFW_SUB_WaitTag: INT := 302;
	cRFW_SUB_SendJob: INT := 304;
	cRFW_SUB_GetData: INT := 306;
	cRFW_SUB_CheckData: INT := 308;
	cRFW_SUB_SendJobTrayID: INT := 310;
	cRFW_SUB_GetDataTrayID: INT := 312;
	cRFW_SUB_CheckDataTrayID: INT := 314;
	cRFW_SUB_Finished: INT := 320;
END_VAR

(*__________________________________________________________________________________________________
¦	
¦	Vistaprint Schweiz GmbH
¦	CH - 8401 Winterthur
¦
¦	www.vistaprint.ch - info@vistaprint.ch
¦___________________________________________________________________________________________________

Function desription:
RFID Reader and Writer
Controlls the communication to the RFID Reader and Writer


History:
Version		Date			Author		Comment
---------------------------------------------------------------------------------------------------
0.00.1		09.07.2013		AVME/PRE	Start history
0.00.2		19.09.2013		AVME/PRE	Implement new Base Concept
0.00.3		24.09.2013		AVME/KVO	Parameter init from element controller to driver
0.00.4		01.10.2013		AVME/PRE	Insert DataChanel to Line
0.00.5		14.11.2013		AVME/PRE	First Checks on the promo machine
___________________________________________________________________________________________________*)


IF (me.bolActivate) AND (pRFD_SIf <>0) THEN // cyclic call enabled
	IF (CIf.Info.bolInitDone=FALSE) THEN // first cycle -> init
		CtrlInit();
		CIf.Info.bolInitDone := TRUE;
	ELSE
		CycleStartDuty();
	
		Always();
		
		StateMachine();
		
		CycleEndDuty();
	END_IF
END_IF;

METHOD PROTECTED Always : BOOL
SUPER^.Always();

// ----------------------------------------------------------------------------------
// cyclic actions outside of statemachine
IF (me.StateMachine.intState<>cSTA_SINGLE_ANSWER) THEN
	pRFD_SIf^.stCur.pData := ADR(SIf.Cur.abytData[0]);
	SIf.Cur.bolPresent := pRFD_SIf^.stStatus.bolPresent;
	IF CIf.Job.bolAlmReset = TRUE THEN
		pRFD_SIf^.stErr.bolErrAck := TRUE;
	END_IF
	fbDtChnToLine_NewRFID.pSIf := ADR(SIf);
	fbDtChnToLine_NewRFID.bolResetError := CIf.Job.bolAlmReset;
	fbDtChnToLine_NewRFID();
	IF fbDtChnToLine_NewRFID.intError <> 0 THEN
		// Set Alarm: SIf.Alm[6].strText := 'Data Channel Error Send Data';
		//pfbAlarmCtrl^.setAlarm(CIf.Info.intCtrlId,6,fbDtChnToLine_NewRFID.intError,ADR(SIf.Alm),E_AlmState.RST,CIf.Job.eMe_ActivAlmClass);	
	END_IF
END_IF

// config driver
pRFD_SIf^.stCfg.bolSimulation := CIf.SwCfg.bolSimulation;
pRFD_SIf^.stCfg.eTyp := SIf.Cfg.eTyp;
pRFD_SIf^.stCfg.stNetId := SIf.Cfg.stNetId; //PLC NetId
pRFD_SIf^.stCfg.uinSlaveAddr := SIf.Cfg.uinSlaveAddr; //Io card Ethercat adress 

// ----------------------------------------------------------------------------------
// Always change actions in Base Library
// ----------------------------------------------------------------------------------
// overrule error always from base -> no EOFF State!! in EOFF go to OFF
IF (me.StateMachine.intStateNext = cSTA_EOFFBusy) THEN
	IF (me.StateMachine.intState=cSTA_OFF) THEN
		me.StateMachine.intStateNext := cSTA_OFF;
	ELSE // stay in OFF
		me.StateMachine.intStateNext := cSTA_OFFBusy;
	END_IF
END_IF

// Conditions Always
IF (((me.Alarm.eActivAlmClass=E_AlmClass.EOFF) OR (me.Alarm.eActivAlmClass=E_AlmClass.OFF) OR (me.intCmd=cCMD_OFF))
		 AND (me.StateMachine.intState<>cSTA_ERROR) AND (me.StateMachine.intState<>cSTA_ERRORQuit) AND
		(me.StateMachine.intState<>cSTA_OFF) AND (me.StateMachine.intState<>cSTA_OFFBusy)) THEN
	// alarm evt EOFF, OFF or cmd off
	me.StateMachine.intStateNext := cSTA_OFFBusy;
END_IF
END_METHOD

METHOD FB_init : BOOL
VAR_INPUT
	///if TRUE, the retain variables are initialized (warm start / cold start)
	bInitRetains: BOOL;
	///if TRUE, the instance afterwards gets moved into the copy code (online change)
	bInCopyCode: BOOL;
END_VAR
VAR
	udiTaskCnt: UDINT;
	ii: UINT;
END_VAR
//------------------------------------------------------------------------------------------------------------------------
// to manually change in new FUB implementation!!!
// define valid commands for this controller
FOR ii:= 0 TO (SIZEOF(CIf.Job.aCmdList)/SIZEOF(CIf.Job.aCmdList[0])-1) BY 1 DO
	IF (CIf.Job.aCmdList[ii].intCmd=cCMD_INITIALIZED) THEN
		// found first empty array element
		EXIT;
	END_IF
END_FOR
CIf.Job.aCmdList[ii].intCmd := RFW_CmdState.cCMD_READ;
CIf.Job.aCmdList[ii].strName := 'Read'; 
CIf.Job.aCmdList[ii].bolAvailable := TRUE;
ii := ii +1;
CIf.Job.aCmdList[ii].intCmd := RFW_CmdState.cCMD_WRITE;
CIf.Job.aCmdList[ii].strName := 'Write';
CIf.Job.aCmdList[ii].bolAvailable := TRUE;
ii := ii +1;
CIf.Job.aCmdList[ii].intCmd := RFW_CmdState.cCMD_ON;
CIf.Job.aCmdList[ii].strName := 'On';
CIf.Job.aCmdList[ii].bolAvailable := TRUE;
ii := ii +1;
CIf.Job.aCmdList[ii].intCmd := cCMD_RUN;
CIf.Job.aCmdList[ii].strName := 'Run';
CIf.Job.aCmdList[ii].bolAvailable := TRUE;

// set name of class/typ
CIf.Info.strType := 'FB_RFID'; 

// set alarm class
SIf.Alm[1].eAlmClass := E_AlmClass.TSTOP;
SIf.Alm[1].strText := 'Communication Error between PLC and RFID Reader'; 
SIf.Alm[2].eAlmClass := E_AlmClass.TSTOP;
SIf.Alm[2].strText := 'Initialisation Error from RFID Reader';
SIf.Alm[3].eAlmClass := E_AlmClass.TSTOP;
SIf.Alm[3].strText := 'RFID Tag Error';
SIf.Alm[4].eAlmClass := E_AlmClass.TSTOP;
SIf.Alm[4].strText := 'timeout wait on Data';
SIf.Alm[5].eAlmClass := E_AlmClass.TSTOP;
SIf.Alm[5].strText := 'Command for this type of RFID not possible';
SIf.Alm[6].eAlmClass := E_AlmClass.INFO;
SIf.Alm[6].strText := 'Data Channel Error Send Data';

//*******************************************************************************
// initial values
//*******************************************************************************

// software configuration
CIf.SwCfg.bolExist := TRUE;
CIf.SwCfg.bolSimulation := FALSE;

// parmeter
SIf.Par.udiReadTime_ms := 30000;
SIf.Par.udiWriteTime_ms := 300000;
SIf.Par.udiMinCmdTime := 100;

// Get correct type
SIf.Cfg.eTyp := E_Typ_RFW.RF382R;
SIf.Cfg.stNetId := '192.168.2.123.1.1'; //PLC NetId
SIf.Cfg.uinSlaveAddr := 1039; //Io card Ethercat adress 
SIf.Cfg.bolGetTrayIDAuto := FALSE;
SIf.Cfg.bolDtChToLine_send := TRUE;
END_METHOD

METHOD PROTECTED getCmdState : STRING
VAR_INPUT
	intCmdState: INT;
	bolState: BOOL;
END_VAR
getCmdState := SUPER^.getCmdState(intCmdState:=intCmdState,bolState:=bolState); // get global/base defined cmds/states
IF (getCmdState='') THEN // global not defined get local
	// get string cmd/state string information in runtime
	IF (bolState=FALSE) THEN
		// cmd's
		CASE intCmdState OF
			RFW_CmdState.cCMD_ON: 
				getCmdState := 'cCMD_ON';
			RFW_CmdState.cCMD_READ: 
				getCmdState := 'cCMD_READ';
			RFW_CmdState.cCMD_WRITE: 
				getCmdState := 'cCMD_WRITE';
		END_CASE;
	ELSE
	
	// cmd's
		CASE intCmdState OF
			RFW_CmdState.cSTA_ONBusy: 
				getCmdState := 'cSTA_ONBusy';
			RFW_CmdState.cSTA_ON: 
				getCmdState := 'cSTA_ON';
			RFW_CmdState.cSTA_READBusy: 
				getCmdState := 'cSTA_READBusy';
			RFW_CmdState.cSTA_READ: 
				getCmdState := 'cSTA_READ';
			RFW_CmdState.cSTA_WRITEBusy: 
				getCmdState := 'cSTA_WRITEBusy';
			RFW_CmdState.cSTA_WRITE: 
				getCmdState := 'cSTA_WRITE';
				
			// SUB States
			cRFW_SUB_WaitTag:
				getCmdState := 'cRFW_SUB_WaitTag';
			cRFW_SUB_SendJob:
				getCmdState := 'cRFW_SUB_SendJob';
			cRFW_SUB_GetData:
				getCmdState := 'cRFW_SUB_GetData';
			cRFW_SUB_CheckData:
				getCmdState := 'cRFW_SUB_CheckData';
			cRFW_SUB_SendJobTrayID:
				getCmdState := 'cRFW_SUB_SendJobTrayID';
			cRFW_SUB_GetDataTrayID:
				getCmdState := 'cRFW_SUB_GetDataTrayID';
			cRFW_SUB_CheckDataTrayID:
				getCmdState := 'cRFW_SUB_CheckDataTrayID';
			cRFW_SUB_Finished: 			
				getCmdState := 'cRFW_SUB_Finished';
		END_CASE;
	END_IF
END_IF
END_METHOD

METHOD getCtrlSIf : POINTER TO T_Ctrl_SIf_RFW
getCtrlSIf := ADR(SIf);
END_METHOD

METHOD PROTECTED IoInBridge : BOOL
// digitale and analoge inputs read from hardware or forcing

IF (CIf.SwCfg.bolSimulation = FALSE) THEN
	;
	//ctrl.In.bol_PosSwitchBasicDefTyp.intern := getInBol(ctrl.ifc.Job.bol_Force ,ADR(ctrl.In.bol_PosSwitchBasicDefTyp);
ELSE
	//simulation of global IO
END_IF
END_METHOD

METHOD PROTECTED IoOutBridge : BOOL
VAR
	bolSwitchValvesOff: BOOL;
END_VAR
// digitale and analoge inputs read from hardware or forcing
IF (CIf.SwCfg.bolSimulation = FALSE) THEN
	// check interlocks to prevent damages
	IF (CIf.Job.bolIlkOverwrite=FALSE) THEN
		;
	END_IF
END_IF
END_METHOD

METHOD PROTECTED sta_ERROR : BOOL
// state implemetation
//--------------------------------------------------------------------------------------
// Entry action
	IF (me.StateMachine.intState<>me.StateMachine.intStateLastCycle) THEN
		me.StateMachine.intStateHistory := me.StateMachine.intStateLastCycle; // -> possibillity to go back to state before error
		me.StateMachine.intStateLastCycle := me.StateMachine.intState;
	END_IF


//--------------------------------------------------------------------------------------
// Cyclic action
	IF (me.StateMachine.intState=me.StateMachine.intStateLastCycle) THEN
		
		IF (pRFD_SIf^.stErr.bolComError = TRUE) OR (pRFD_SIf^.stErr.bolProtcolError = TRUE) THEN
			// SIf.Alm[1].strText := 'Communication Error between PLC and RFID Reader'; 
			pfbAlarmCtrl^.setAlarm(CIf.Info.intCtrlId,1,UDINT_TO_DINT(pRFD_SIf^.stErr.udiErrorID),ADR(SIf.Alm),E_AlmState.RST,CIf.Job.eMe_ActivAlmClass);
		ELSIF pRFD_SIf^.stErr.bolSDOError = TRUE THEN
			// SIf.Alm[2].strText := 'Initialisation Error from RFID Reader';
			pfbAlarmCtrl^.setAlarm(CIf.Info.intCtrlId,2,UDINT_TO_DINT(pRFD_SIf^.stErr.udiErrorID),ADR(SIf.Alm),E_AlmState.RST,CIf.Job.eMe_ActivAlmClass);
		ELSIF (pRFD_SIf^.stErr.bolRFIDError = TRUE) THEN
			// SIf.Alm[3].strText := 'RFID Tag Error';
			pfbAlarmCtrl^.setAlarm(CIf.Info.intCtrlId,3,UDINT_TO_DINT(pRFD_SIf^.stErr.udiErrorID),ADR(SIf.Alm),E_AlmState.RST,CIf.Job.eMe_ActivAlmClass);
		END_IF
		
		
		// State Change Condition
		IF (CIf.Job.bolAlmReset = TRUE) THEN
			me.StateMachine.intStateNext := cSTA_ERRORQuit;
		END_IF
	END_IF




//--------------------------------------------------------------------------------------
// Exit action
	IF (me.StateMachine.intState<>me.StateMachine.intStateNext) THEN
		IF 	CIf.Job.intACmd > cCMD_OFF THEN
			CIf.Job.intACmd := cCMD_DONE;
		END_IF

	END_IF
END_METHOD

METHOD PROTECTED sta_OFF : BOOL
// state implemetation
//--------------------------------------------------------------------------------------
// Entry action
	IF (me.StateMachine.intState<>me.StateMachine.intStateLastCycle) THEN
		me.StateMachine.intStateLastCycle := me.StateMachine.intState;
		
	END_IF


//--------------------------------------------------------------------------------------
// Cyclic action
	IF (me.StateMachine.intState=me.StateMachine.intStateLastCycle) THEN
		
		;
		
		
		// State Change Condition
		IF (me.Alarm.eActivAlmClass<>E_AlmClass.EOFF) AND (me.Alarm.eActivAlmClass<>E_AlmClass.OFF) THEN
			IF(me.intCmd=cCMD_RUN) THEN
				me.StateMachine.intStateNext := cSTA_RUNBusy;
			ELSIF ((me.intCmd=RFW_CmdState.cCMD_READ) OR (me.intCmd=RFW_CmdState.cCMD_WRITE)) AND (SIf.Cfg.eTyp = E_Typ_RFW.RF382R) THEN
				// SIf.Alm[5].strText := 'Command for this type of RFID not possible';
				pfbAlarmCtrl^.setAlarm(CIf.Info.intCtrlId,5,UDINT_TO_DINT(pRFD_SIf^.stErr.udiErrorID),ADR(SIf.Alm),E_AlmState.RST,CIf.Job.eMe_ActivAlmClass);			
			ELSIF(me.intCmd=RFW_CmdState.cCMD_READ) THEN
				me.StateMachine.intStateNext := RFW_CmdState.cSTA_READBusy;
			ELSIF(me.intCmd=RFW_CmdState.cCMD_WRITE) THEN
				me.StateMachine.intStateNext := RFW_CmdState.cSTA_WRITEBusy;
			ELSIF(me.intCmd=RFW_CmdState.cCMD_ON) THEN
				me.StateMachine.intStateNext := RFW_CmdState.cSTA_ONBusy;			
			END_IF
		END_IF
	END_IF




//--------------------------------------------------------------------------------------
// Exit action
	IF (me.StateMachine.intState<>me.StateMachine.intStateNext) THEN
		;
	END_IF
END_METHOD

METHOD PROTECTED sta_OFFBusy : BOOL
// state implemetation
//--------------------------------------------------------------------------------------
// Entry action
	IF (me.StateMachine.intState<>me.StateMachine.intStateLastCycle) THEN
		me.StateMachine.intStateLastCycle := me.StateMachine.intState;
		fbSimulationTimer.IN := FALSE;
		fbSimulationTimer.PT := UDINT_TO_TIME(SIf.Par.udiReadTime_ms / 2);
		fbSimulationTimer(); // set time/reset timer
		fbSimulationTimer.IN := TRUE; // start timer
		
	END_IF


//--------------------------------------------------------------------------------------
// Cyclic action
	IF (me.StateMachine.intState=me.StateMachine.intStateLastCycle) THEN
		// Simulation
		IF (CIf.SwCfg.bolSimulation) THEN
			fbSimulationTimer(); // simulation time
			IF (fbSimulationTimer.Q) THEN
				pRFD_SIf^.intCmd := RFD_Cmd.cRFD_CMD_DONE;
				SIf.Cur.bolPresent := FALSE;
			END_IF
		END_IF
		
	
		// State Change Condition
		IF pRFD_SIf^.stErr.bolErrorActive = TRUE THEN // AND (me.StateMachine.udiTimeInState_ms>SIf.Par.udiWriteTime_ms) 
			me.StateMachine.intStateNext :=  cSTA_ERROR;
		//ELSIF(pRFD_SIf^.intCmd = RFD_Cmd.cRFD_CMD_DONE) THEN
		ELSIF (TRUE) THEN
			me.StateMachine.intStateNext := cSTA_OFF;
		END_IF
	END_IF




//--------------------------------------------------------------------------------------
// Exit action
	IF (me.StateMachine.intState<>me.StateMachine.intStateNext) THEN
		;
	END_IF
END_METHOD

METHOD PROTECTED sta_ON : BOOL
// state implemetation
//--------------------------------------------------------------------------------------
// Entry action
	IF (me.StateMachine.intState<>me.StateMachine.intStateLastCycle) THEN
		me.StateMachine.intStateLastCycle := me.StateMachine.intState;
		bolNewTag := FALSE;
		me.SubStateMachine.intState := cRFW_SUB_WaitTag-1; // init first state - string
		me.SubStateMachine.intStateNext := cRFW_SUB_WaitTag;
		fbSimulationTimer.IN := FALSE;
		fbSimulationTimer.PT := UDINT_TO_TIME(SIf.Par.udiReadTime_ms / 2);
		fbSimulationTimer(); // set time/reset timer
		fbSimulationTimer.IN := TRUE; // start timer
		
	END_IF


//--------------------------------------------------------------------------------------
// Cyclic action
	IF (me.StateMachine.intState=me.StateMachine.intStateLastCycle) THEN

		// Simulation
		
		// Function
				
		// State Change Condition
		IF (pRFD_SIf^.stErr.bolErrorActive = TRUE) THEN  
			me.StateMachine.intStateNext :=  cSTA_ERROR;
		ELSIF ((me.intCmd=cCMD_READ) OR (me.intCmd=cCMD_WRITE)) AND (SIf.Cfg.eTyp = E_Typ_RFW.RF382R) THEN
			// SIf.Alm[5].strText := 'Command for this type of RFID not possible';
			pfbAlarmCtrl^.setAlarm(CIf.Info.intCtrlId,5,UDINT_TO_DINT(pRFD_SIf^.stErr.udiErrorID),ADR(SIf.Alm),E_AlmState.RST,CIf.Job.eMe_ActivAlmClass);			
		ELSIF (me.intCmd=cCMD_READ) THEN
			me.StateMachine.intStateNext := cSTA_READBusy;
		ELSIF(me.intCmd=cCMD_WRITE) THEN
			me.StateMachine.intStateNext := cSTA_WRITEBusy;
		ELSIF(me.intCmd=cCMD_RUN) THEN
			me.StateMachine.intStateNext := cSTA_RUNBusy;			
		END_IF
	END_IF




//--------------------------------------------------------------------------------------
// Exit action
	IF (me.StateMachine.intState<>me.StateMachine.intStateNext) THEN
		;		
	END_IF
END_METHOD

METHOD PROTECTED sta_ONbusy : BOOL
// state implemetation
//--------------------------------------------------------------------------------------
// Entry action
	IF (me.StateMachine.intState<>me.StateMachine.intStateLastCycle) THEN
		me.StateMachine.intStateLastCycle := me.StateMachine.intState;
		bolNewTag := FALSE;
		me.SubStateMachine.intState := cRFW_SUB_WaitTag;
		SIf.Cur.dwoJob := RFID_Data.cRFID_TrayID;
		
		fbSimulationTimer.IN := FALSE;
		fbSimulationTimer.PT := UDINT_TO_TIME(SIf.Par.udiReadTime_ms / 2);
		fbSimulationTimer(); // set time/reset timer
		fbSimulationTimer.IN := TRUE; // start timer
		
	END_IF


//--------------------------------------------------------------------------------------
// Cyclic action
	IF (me.StateMachine.intState=me.StateMachine.intStateLastCycle) THEN

		// Simulation
		IF (CIf.SwCfg.bolSimulation) THEN
			pRFD_SIf^.stStatus.bolOn := TRUE;
			fbSimulationTimer(); // simulation time
			IF (fbSimulationTimer.Q) THEN
				;
			END_IF
		END_IF
		
		// Function
		IF(pRFD_SIf^.stStatus.bolOn = FALSE) THEN
			pRFD_SIf^.intCmd := RFD_Cmd.cRFD_CMD_CTRL_ON;
		END_IF
		
		// State Change Condition
		IF (pRFD_SIf^.stErr.bolErrorActive = TRUE) THEN  
			me.StateMachine.intStateNext :=  cSTA_ERROR;
		ELSIF(pRFD_SIf^.stStatus.bolOn = TRUE) THEN
			me.StateMachine.intStateNext := RFW_CmdState.cSTA_ON;
		END_IF
	END_IF




//--------------------------------------------------------------------------------------
// Exit action
	IF (me.StateMachine.intState<>me.StateMachine.intStateNext) THEN
		;		
	END_IF
END_METHOD

METHOD PROTECTED sta_PON : BOOL
// state implemetation
//--------------------------------------------------------------------------------------
// Entry action
	IF (me.StateMachine.intState<>me.StateMachine.intStateLastCycle) THEN
		me.StateMachine.intStateLastCycle := me.StateMachine.intState;
		
	END_IF


//--------------------------------------------------------------------------------------
// Cyclic action
	IF (me.StateMachine.intState=me.StateMachine.intStateLastCycle) THEN
		
		;
		
		
		// State Change Condition
		IF (me.intCmd<>cCMD_PON) AND (me.intCmd<>cCMD_DONE) THEN
			me.StateMachine.intStateNext := cSTA_OFFBusy;
		END_IF
	END_IF




//--------------------------------------------------------------------------------------
// Exit action
	IF (me.StateMachine.intState<>me.StateMachine.intStateNext) THEN
		;
	END_IF
END_METHOD

METHOD PROTECTED sta_PONBusy : BOOL
// state implemetation
//--------------------------------------------------------------------------------------
// Entry action
	IF (me.StateMachine.intState<>me.StateMachine.intStateLastCycle) THEN
		me.StateMachine.intStateLastCycle := me.StateMachine.intState;
		fbSimulationTimer.IN := FALSE;
		fbSimulationTimer.PT := UDINT_TO_TIME(SIf.Par.udiReadTime_ms / 2);
		fbSimulationTimer(); // set time/reset timer
		fbSimulationTimer.IN := TRUE; // start timer
		
		IF (CIf.SwCfg.bolSimulation = FALSE) THEN
			pRFD_SIf^.intCmd := RFD_Cmd.cRFD_CMD_CTRL_ON; // parameter initialisation on driver
		END_IF
	END_IF


//--------------------------------------------------------------------------------------
// Cyclic action
	IF (me.StateMachine.intState=me.StateMachine.intStateLastCycle) THEN
		// Simulation
		IF (CIf.SwCfg.bolSimulation) THEN
			fbSimulationTimer(); // simulation time
			IF (fbSimulationTimer.Q) THEN
				pRFD_SIf^.intCmd := RFD_Cmd.cRFD_CMD_DONE;
				SIf.Cur.bolPresent := FALSE;
			END_IF
		END_IF
		
	
		// State Change Condition
		IF (pRFD_SIf^.stErr.bolErrorActive = TRUE) AND (CIf.SwCfg.bolSimulation = FALSE) THEN // AND (me.StateMachine.udiTimeInState_ms>SIf.Par.udiWriteTime_ms) 
			me.StateMachine.intStateNext :=  cSTA_ERROR;
		ELSIF (pRFD_SIf^.intCmd = RFD_Cmd.cRFD_CMD_DONE) THEN
			me.StateMachine.intStateNext := cSTA_PON;
		END_IF
	END_IF




//--------------------------------------------------------------------------------------
// Exit action
	IF (me.StateMachine.intState<>me.StateMachine.intStateNext) THEN
		;
	END_IF
END_METHOD

METHOD PROTECTED sta_READ : BOOL
// state implemetation
//--------------------------------------------------------------------------------------
// Entry action
	IF (me.StateMachine.intState<>me.StateMachine.intStateLastCycle) THEN
		me.StateMachine.intStateLastCycle := me.StateMachine.intState;

	END_IF


//--------------------------------------------------------------------------------------
// Cyclic action
	IF (me.StateMachine.intState=me.StateMachine.intStateLastCycle) THEN

		// Simulation
		IF (CIf.SwCfg.bolSimulation) THEN
			;
		END_IF
		
		// State Change Condition
		IF(me.intCmd=cCMD_RUN) THEN
			me.StateMachine.intStateNext := cSTA_RUNBusy;
		ELSIF ((me.intCmd=RFW_CmdState.cCMD_READ) OR (me.intCmd=RFW_CmdState.cCMD_WRITE)) AND (SIf.Cfg.eTyp = E_Typ_RFW.RF382R) THEN
			// SIf.Alm[5].strText := 'Command for this type of RFID not possible';
			pfbAlarmCtrl^.setAlarm(CIf.Info.intCtrlId,5,UDINT_TO_DINT(pRFD_SIf^.stErr.udiErrorID),ADR(SIf.Alm),E_AlmState.RST,CIf.Job.eMe_ActivAlmClass);			
		ELSIF(me.intCmd=RFW_CmdState.cCMD_WRITE) THEN
			me.StateMachine.intStateNext := RFW_CmdState.cSTA_WRITEBusy;
		ELSIF(me.intCmd=RFW_CmdState.cCMD_READ) THEN
			me.StateMachine.intStateNext := RFW_CmdState.cSTA_READBusy;
		ELSIF(me.intCmd=RFW_CmdState.cCMD_ON) THEN
			me.StateMachine.intStateNext := RFW_CmdState.cSTA_ONBusy;			
		END_IF
	END_IF




//--------------------------------------------------------------------------------------
// Exit action
	IF (me.StateMachine.intState<>me.StateMachine.intStateNext) THEN
		;
	END_IF
END_METHOD

METHOD PROTECTED sta_READBusy : BOOL
// state implemetation
//--------------------------------------------------------------------------------------
// Entry action
	IF (me.StateMachine.intState<>me.StateMachine.intStateLastCycle) THEN
		me.StateMachine.intStateLastCycle := me.StateMachine.intState;
		
		fbSimulationTimer.IN := FALSE;
		fbSimulationTimer.PT := UDINT_TO_TIME(SIf.Par.udiReadTime_ms / 2);
		fbSimulationTimer(); // set time/reset timer
		fbSimulationTimer.IN := TRUE; // start timer
		
		IF SIf.Cur.dwoJob = 0 THEN
			SIf.Cur.dwoJob := RFID_Data.cRFID_AllData;
		END_IF
		
		bolAllFinished := FALSE;
		dwoJobIntern := SIf.Cur.dwoJob;
		
		uinDataAdress := DWORD_TO_UINT(dwoJobIntern);
		uinDataAdress := uinDataAdress MOD 16#100;							// Maximum 255 data
		
		pRFD_SIf^.stCur.uinAdressData := uinDataAdress;
		pRFD_SIf^.stCur.uinAdressTag := DWORD_TO_UINT(dwoJobIntern);
		pRFD_SIf^.stCur.usiCount := DWORD_TO_USINT(SHR(dwoJobIntern,16));
		
		udiTimeDelayRead := 0;

		IF (CIf.SwCfg.bolSimulation = FALSE) THEN
			pRFD_SIf^.intCmd := RFD_Cmd.cRFD_CMD_Read;
		END_IF
	END_IF


//--------------------------------------------------------------------------------------
// Cyclic action
	IF (me.StateMachine.intState=me.StateMachine.intStateLastCycle) THEN

		// Simulation
		IF (CIf.SwCfg.bolSimulation) THEN
			fbSimulationTimer(); // simulation time
			IF (fbSimulationTimer.Q) THEN
				pRFD_SIf^.intCmd := RFD_Cmd.cRFD_CMD_DONE;
			END_IF
		END_IF
		
		// Function
		// By Read all the Tray ID has to be readed too
		IF (pRFD_SIf^.intCmd = RFD_Cmd.cRFD_CMD_DONE) AND (udiTimeDelayRead > SIf.Par.udiMinCmdTime) THEN
		//---------------------------------------
			udiTimeDelayRead := 0;
			// Prepare Data from read memory
			// Repetition ID
			IF (dwoJobIntern = RFID_Data.cRFID_AllData) OR (dwoJobIntern = RFID_Data.cRFID_RepetionID) THEN
				uinDataAdress := DWORD_TO_UINT(RFID_Data.cRFID_RepetionID);
				uinDataAdress := uinDataAdress  MOD 16#100;							// only 0..255
				IF ((uinDataAdress >= 0) AND (uinDataAdress <= 255)) THEN
					SIf.Cur.stData.usiRepetitionID := SIf.Cur.abytData[uinDataAdress];
				END_IF
			END_IF
			// Tray Info
			IF (dwoJobIntern = RFID_Data.cRFID_AllData) OR (dwoJobIntern = RFID_Data.cRFID_TrayInfo) THEN
				uinDataAdress := DWORD_TO_UINT(RFID_Data.cRFID_TrayInfo);
				uinDataAdress := uinDataAdress  MOD 16#100;							// only 0..255
				IF ((uinDataAdress >= 0) AND (uinDataAdress <= 255)) THEN
					SIf.Cur.stData.bolWorkstation2 := SIf.Cur.abytData[uinDataAdress].0;
					SIf.Cur.stData.bolDeleteFileAfterPrint := SIf.Cur.abytData[uinDataAdress].6;
					SIf.Cur.stData.bolPrintOk := SIf.Cur.abytData[uinDataAdress].7;
				END_IF
			END_IF
			// Height of tray
			IF (dwoJobIntern = RFID_Data.cRFID_AllData) OR (dwoJobIntern = RFID_Data.cRFID_HeighOfTray) THEN
				uinDataAdress := DWORD_TO_UINT(RFID_Data.cRFID_HeighOfTray);
				uinDataAdress := uinDataAdress  MOD 16#100;							// only 0..255
				IF ((uinDataAdress >= 0) AND (uinDataAdress <= 255)) THEN
					SIf.Cur.stData.bolHeightUseMeasure := SIf.Cur.abytData[uinDataAdress].0;
					SIf.Cur.stData.usiHeightOffset := 0;
					SIf.Cur.stData.usiHeightOffset.0 := SIf.Cur.abytData[uinDataAdress].1;
					SIf.Cur.stData.usiHeightOffset.1 := SIf.Cur.abytData[uinDataAdress].2;
					SIf.Cur.stData.usiHeightOffset.2 := SIf.Cur.abytData[uinDataAdress].3;
					SIf.Cur.stData.bolHeightOffsetSignMinus := SIf.Cur.abytData[uinDataAdress].4;
				END_IF
			END_IF
			// Pretreatment
			IF (dwoJobIntern = RFID_Data.cRFID_AllData) OR (dwoJobIntern = RFID_Data.cRFID_RepetionID) THEN
				uinDataAdress := DWORD_TO_UINT(RFID_Data.cRFID_Pretreatment);
				uinDataAdress := uinDataAdress  MOD 16#100;							// only 0..255
				IF ((uinDataAdress >= 0) AND (uinDataAdress <= 255)) THEN
					SIf.Cur.stData.bolIonizer := SIf.Cur.abytData[uinDataAdress].1;
					SIf.Cur.stData.usiPlasmaLevel := 0;
					SIf.Cur.stData.usiPlasmaLevel.0 := SIf.Cur.abytData[uinDataAdress].2;
					SIf.Cur.stData.usiPlasmaLevel.1 := SIf.Cur.abytData[uinDataAdress].3;
					SIf.Cur.stData.bolPrintPass := SIf.Cur.abytData[uinDataAdress].4;
					SIf.Cur.stData.bolNozzleCheck := SIf.Cur.abytData[uinDataAdress].5;
					SIf.Cur.stData.bolAligneCheck := SIf.Cur.abytData[uinDataAdress].6;
				END_IF
			END_IF
			// UV-curing
			IF (dwoJobIntern = RFID_Data.cRFID_AllData) OR (dwoJobIntern = RFID_Data.cRFID_UVcuring) THEN
				uinDataAdress := DWORD_TO_UINT(RFID_Data.cRFID_UVcuring);
				uinDataAdress := uinDataAdress  MOD 16#100;							// only 0..255
				IF ((uinDataAdress >= 0) AND (uinDataAdress <= 255)) THEN
					SIf.Cur.stData.usiUVPinningLevel := 0;
					SIf.Cur.stData.usiUVPinningLevel.0 := SIf.Cur.abytData[uinDataAdress].0;
					SIf.Cur.stData.usiUVPinningLevel.1 := SIf.Cur.abytData[uinDataAdress].1;
					SIf.Cur.stData.usiUVPinningLevel.2 := SIf.Cur.abytData[uinDataAdress].2;
					SIf.Cur.stData.usiUVPinningLevel.3 := SIf.Cur.abytData[uinDataAdress].3;
		
					SIf.Cur.stData.usiUVLampLevel := 0;
					SIf.Cur.stData.usiUVLampLevel.0 := SIf.Cur.abytData[uinDataAdress].4;
					SIf.Cur.stData.usiUVLampLevel.1 := SIf.Cur.abytData[uinDataAdress].5;
					SIf.Cur.stData.usiUVLampLevel.2 := SIf.Cur.abytData[uinDataAdress].6;
					SIf.Cur.stData.usiUVLampLevel.3 := SIf.Cur.abytData[uinDataAdress].7;
				END_IF
			END_IF
			// Filename
			IF (dwoJobIntern = RFID_Data.cRFID_AllData) OR (dwoJobIntern = RFID_Data.cRFID_Filename) THEN
				uinDataAdress := DWORD_TO_UINT(RFID_Data.cRFID_Filename);
				uinDataLengh := DWORD_TO_UINT(SHR(RFID_Data.cRFID_Filename,16));
				uinDataAdress := uinDataAdress  MOD 16#100;							// only 0..255
				IF ((uinDataAdress >= 0) AND (uinDataAdress <= 255)) THEN
					strTemp := USINT_TO_STRING(SIf.Cur.abytData[uinDataAdress]);
					strTemp := TC2_STANDARD.CONCAT('-', strTemp);
					uliTemp := 0;
					uinDataAdress := uinDataAdress+1;	// Next signs
					Tc2_System.MEMCPY(destAddr := ADR(uliTemp), srcAddr := ADR(SIf.Cur.abytData[uinDataAdress]), n:= (uinDataLengh-1));
		
					SIf.Cur.stData.strFileName := TC2_STANDARD.CONCAT(ULINT_TO_STRING(uliTemp), strTemp);
				END_IF
			END_IF
			// Brush
			IF (dwoJobIntern = RFID_Data.cRFID_AllData) OR (dwoJobIntern = RFID_Data.cRFID_Brush) THEN
				uinDataAdress := DWORD_TO_UINT(RFID_Data.cRFID_Brush);
				uinDataAdress := uinDataAdress  MOD 16#100;							// only 0..255
				IF ((uinDataAdress >= 0) AND (uinDataAdress <= 255)) THEN
					SIf.Cur.stData.bolBrush := SIf.Cur.abytData[uinDataAdress].0;
					SIf.Cur.stData.bolBrushClean := SIf.Cur.abytData[uinDataAdress].1;
					SIf.Cur.stData.bolBrushFans := SIf.Cur.abytData[uinDataAdress].2;
					SIf.Cur.stData.bolGutterClean := SIf.Cur.abytData[uinDataAdress].6;
					SIf.Cur.stData.bolSpecialTray := SIf.Cur.abytData[uinDataAdress].7;
				END_IF
			END_IF
			
			// Tray ID
			IF (dwoJobIntern = RFID_Data.cRFID_TrayID) THEN
				uinDataAdress := DWORD_TO_UINT(RFID_Data.cRFID_TrayID);
				uinDataAdress := uinDataAdress  MOD 16#100;							// only 0..255
				IF ((uinDataAdress >= 0) AND (uinDataAdress <= 255)) THEN
					uinDataLengh := DWORD_TO_UINT(SHR(RFID_Data.cRFID_TrayID,16));
					SIf.Cur.stData.strTrayID := '';
					udiTemp := Tc2_System.MEMCPY(destAddr:=ADR(SIf.Cur.stData.strTrayID), srcAddr:=ADR(SIf.Cur.abytData[uinDataAdress]), n:=uinDataLengh);
				END_IF
			END_IF
	
			// Tag ID
			IF (dwoJobIntern = RFID_Data.cRFID_TagID) THEN
				uinDataAdress := DWORD_TO_UINT(RFID_Data.cRFID_TagID);
				uinDataAdress := uinDataAdress  MOD 16#100;							// only 0..255
				IF ((uinDataAdress >= 0) AND (uinDataAdress <= 255)) THEN
					uinDataLengh := DWORD_TO_UINT(SHR(RFID_Data.cRFID_TagID,16));
					SIf.Cur.stData.strTagID := '';
					udiTemp := Tc2_System.MEMCPY(destAddr:=ADR(SIf.Cur.stData.uliTagID), srcAddr:=ADR(pRFD_SIf^.stStatus.abyteUID), n:=8);
					SIf.Cur.stData.strTagID := FB_ULINT_TO_HEXSTRING(in_uliValue:= SIf.Cur.stData.uliTagID);	
				END_IF
			END_IF	
		//---------------------------------------
		//END_IF
			IF SIf.Cur.dwoJob = RFID_Data.cRFID_AllData THEN
				//IF udiTimeDelayRead >= 100 THEN // Wait 100ms
					IF dwoJobIntern = RFID_Data.cRFID_AllData THEN
						dwoJobIntern := RFID_Data.cRFID_TrayID;
						uinDataAdress := DWORD_TO_UINT(dwoJobIntern);
						uinDataAdress := uinDataAdress MOD 16#100;							// Maximum 255 data
						
						pRFD_SIf^.stCur.uinAdressData := uinDataAdress;
						pRFD_SIf^.stCur.uinAdressTag := DWORD_TO_UINT(dwoJobIntern);
						pRFD_SIf^.stCur.usiCount := DWORD_TO_USINT(SHR(dwoJobIntern,16));
				
						pRFD_SIf^.intCmd := RFD_Cmd.cRFD_CMD_Read;
						udiTimeDelayRead := 0;
					ELSIF dwoJobIntern = RFID_Data.cRFID_TrayID THEN
						dwoJobIntern := RFID_Data.cRFID_TagID;
						uinDataAdress := DWORD_TO_UINT(dwoJobIntern);
						uinDataAdress := uinDataAdress MOD 16#100;							// Maximum 255 data
						
						pRFD_SIf^.stCur.uinAdressData := uinDataAdress;
						pRFD_SIf^.stCur.uinAdressTag := DWORD_TO_UINT(dwoJobIntern);
						pRFD_SIf^.stCur.usiCount := DWORD_TO_USINT(SHR(dwoJobIntern,16));
				
						pRFD_SIf^.intCmd := RFD_Cmd.cRFD_CMD_MDS;
						udiTimeDelayRead := 0;
					ELSE
						bolAllFinished := TRUE;
					END_IF
				//ELSE
					udiTimeDelayRead := udiTimeDelayRead + me.FUBInfo.udiSample_ms;			
				//END_IF
			ELSE
				bolAllFinished := TRUE;
			END_IF
		END_IF
		// State Change Condition
		IF (pRFD_SIf^.stErr.bolErrorActive = TRUE) THEN  
			me.StateMachine.intStateNext :=  cSTA_ERROR;
		ELSIF (me.StateMachine.udiTimeInState_ms > SIf.Par.udiWriteTime_ms) THEN
			// SIf.Alm[4].strText := 'timeout wait on Data';
			pfbAlarmCtrl^.setAlarm(CIf.Info.intCtrlId,4,0,ADR(SIf.Alm),E_AlmState.RST,CIf.Job.eMe_ActivAlmClass);
			me.StateMachine.intStateNext :=  cSTA_ERROR;
		ELSIF (bolAllFinished = TRUE) THEN
			me.StateMachine.intStateNext := cSTA_READ;
		END_IF
	END_IF

	udiTimeDelayRead := udiTimeDelayRead + me.FUBInfo.udiSample_ms;



//--------------------------------------------------------------------------------------
// Exit action
	IF (me.StateMachine.intState<>me.StateMachine.intStateNext) THEN
		;
	END_IF
END_METHOD

METHOD PROTECTED sta_RUN : BOOL
// state implemetation
//--------------------------------------------------------------------------------------
// Entry action
	IF (me.StateMachine.intState<>me.StateMachine.intStateLastCycle) THEN
		me.StateMachine.intStateLastCycle := me.StateMachine.intState;
		bolNewTag := FALSE;
		me.SubStateMachine.intState := cRFW_SUB_WaitTag-1; // init first state - string
		me.SubStateMachine.intStateNext := cRFW_SUB_WaitTag;
		fbSimulationTimer.IN := FALSE;
		fbSimulationTimer.PT := UDINT_TO_TIME(SIf.Par.udiReadTime_ms / 2);
		fbSimulationTimer(); // set time/reset timer
		fbSimulationTimer.IN := TRUE; // start timer
		
	END_IF


//--------------------------------------------------------------------------------------
// Cyclic action
	IF (me.StateMachine.intState=me.StateMachine.intStateLastCycle) THEN

		// Simulation
		IF (CIf.SwCfg.bolSimulation) THEN
			fbSimulationTimer(); // simulation time
			IF (fbSimulationTimer.IN = FALSE) THEN
				fbSimulationTimer.IN := TRUE;
			END_IF
			IF pRFD_SIf^.intCmd <> RFD_Cmd.cRFD_CMD_DONE THEN
				pRFD_SIf^.intCmd := RFD_Cmd.cRFD_CMD_DONE;
			END_IF
			IF (fbSimulationTimer.Q) THEN
				fbSimulationTimer.IN := FALSE;
				IF SIf.Cur.bolPresent = FALSE THEN
					SIf.Cur.bolPresent := TRUE;
					SIf.Cur.stData.uliTagID := SIf.Cur.stData.uliTagID + 1;
					Tc2_System.MEMCPY(destAddr:=ADR(pRFD_SIf^.stStatus.abyteUID), srcAddr:=ADR(SIf.Cur.stData.uliTagID), n:=8);
				ELSE
					SIf.Cur.bolPresent := FALSE;
				END_IF
			END_IF
		END_IF
		
		// Function
		// If the RF ID Reader does not send automatically the Tag ID, read it if a new Tag is ready
		IF (SIf.Cfg.eTyp = E_Typ_RFW.RF310R) AND (CIf.SwCfg.bolSimulation = FALSE) THEN
			IF ((SIf.Cur.bolPresent = TRUE) AND (bolRENewTag = FALSE)) THEN
				bolNewTag := TRUE;
				bolRENewTag := TRUE;
			ELSIF (SIf.Cur.bolPresent = FALSE) THEN
				bolRENewTag := FALSE;
				bolNewTag := FALSE;
			END_IF
			
			//--------------------------------------------------------------------------------------
			// sub state machine for sequence
			CASE me.SubStateMachine.intState OF
				//--------------------------------------------------------------------------------------
				cRFW_SUB_WaitTag:
					IF (bolNewTag = TRUE) THEN
						me.SubStateMachine.intStateNext := cRFW_SUB_SendJob;
					END_IF
				
				cRFW_SUB_SendJob:
					pRFD_SIf^.stCur.uinAdressData :=0;
					pRFD_SIf^.stCur.uinAdressTag := DWORD_TO_UINT(RFID_Data.cRFID_TagID);
					pRFD_SIf^.stCur.usiCount := DWORD_TO_USINT(SHR(RFID_Data.cRFID_TagID,16));
				
					pRFD_SIf^.intCmd := RFD_Cmd.cRFD_CMD_MDS;
					
					me.SubStateMachine.intStateNext := cRFW_SUB_GetData;
					
				cRFW_SUB_GetData:
					IF pRFD_SIf^.intCmd = RFD_Cmd.cRFD_CMD_DONE THEN
						me.SubStateMachine.intStateNext := cRFW_SUB_CheckData;
					END_IF
				
				cRFW_SUB_CheckData:
					SIf.Cur.stData.strTagID := '';
					Tc2_System.MEMCPY(destAddr:=ADR(SIf.Cur.stData.uliTagID), srcAddr:=ADR(pRFD_SIf^.stStatus.abyteUID), n:=8);
					SIf.Cur.stData.strTagID := FB_ULINT_TO_HEXSTRING(in_uliValue:= SIf.Cur.stData.uliTagID);	

					IF (SIf.Cfg.bolGetTrayIDAuto = TRUE) THEN
						me.SubStateMachine.intStateNext := cRFW_SUB_SendJobTrayID;
					ELSE
						me.SubStateMachine.intStateNext := cRFW_SUB_Finished;
					END_IF
					
				cRFW_SUB_SendJobTrayID:
					uinDataAdress := DWORD_TO_UINT(RFID_Data.cRFID_TrayID);
					uinDataAdress := uinDataAdress MOD 16#100;							// Maximum 255 data
					uinDataLengh := DWORD_TO_UINT(SHR(RFID_Data.cRFID_TrayID,16));
					pRFD_SIf^.stCur.uinAdressData :=uinDataAdress;
					pRFD_SIf^.stCur.uinAdressTag := DWORD_TO_UINT(RFID_Data.cRFID_TrayID);
					pRFD_SIf^.stCur.usiCount := DWORD_TO_USINT(SHR(RFID_Data.cRFID_TrayID,16));
				
					pRFD_SIf^.intCmd := RFD_Cmd.cRFD_CMD_Read;
					
					me.SubStateMachine.intStateNext := cRFW_SUB_GetData;
					
				cRFW_SUB_GetDataTrayID:
					IF pRFD_SIf^.intCmd = RFD_Cmd.cRFD_CMD_DONE THEN
						me.SubStateMachine.intStateNext := cRFW_SUB_CheckData;
					END_IF
				
				cRFW_SUB_CheckDataTrayID:
					uinDataAdress := DWORD_TO_UINT(RFID_Data.cRFID_TrayID);
					uinDataAdress := uinDataAdress MOD 16#100;							// Maximum 255 data
					uinDataLengh := DWORD_TO_UINT(SHR(RFID_Data.cRFID_TrayID,16));
					SIf.Cur.stData.strTagID := '';
					Tc2_System.MEMCPY(destAddr:=ADR(SIf.Cur.stData.strTrayID), srcAddr:=ADR(pRFD_SIf^.stStatus.abyteUID[uinDataAdress]), n:=uinDataLengh);

					me.SubStateMachine.intStateNext := cRFW_SUB_Finished;
	
				cRFW_SUB_Finished:
					bolNewTag := FALSE;				
					me.SubStateMachine.intStateNext := cRFW_SUB_WaitTag;
					
			END_CASE
		ELSIF (SIf.Cfg.eTyp = E_Typ_RFW.RF382R) THEN
			SIf.Cur.stData.strTagID := '';
			Tc2_System.MEMCPY(destAddr:=ADR(SIf.Cur.stData.uliTagID), srcAddr:=ADR(pRFD_SIf^.stStatus.abyteUID), n:=8);
			SIf.Cur.stData.strTagID := FB_ULINT_TO_HEXSTRING(in_uliValue:= SIf.Cur.stData.uliTagID);	
			
		END_IF
		
		IF uliTagID_old <> SIf.Cur.stData.uliTagID THEN
			IF SIf.Cfg.bolDtChToLine_send = TRUE THEN
				IF SIf.Cfg.bolGetTrayIDAuto THEN
					intDtChnToLineState	:= fbDtChnToLine_NewRFID.Creat(In_uliTagID:= SIf.Cur.stData.uliTagID, In_strID:= SIf.Cur.stData.strTrayID);
				ELSE
					intDtChnToLineState	:= fbDtChnToLine_NewRFID.Creat(In_uliTagID:= SIf.Cur.stData.uliTagID, In_strID:= SIf.Cur.stData.strTagID);						
				END_IF
				IF intDtChnToLineState >= 0 THEN
					uliTagID_old := SIf.Cur.stData.uliTagID;
				ELSE
					// Set Alarm: SIf.Alm[6].strText := 'Data Channel Error Send Data';
					//pfbAlarmCtrl^.setAlarm(CIf.Info.intCtrlId,6,intDtChnToLineState,ADR(SIf.Alm),E_AlmState.RST,CIf.Job.eMe_ActivAlmClass);					
				END_IF
			ELSE
				uliTagID_old := SIf.Cur.stData.uliTagID;
			END_IF		
		END_IF
		
				
		// State Change Condition
		IF (pRFD_SIf^.stErr.bolErrorActive = TRUE) THEN  
			me.StateMachine.intStateNext :=  cSTA_ERROR;
		ELSIF ((me.intCmd=RFW_CmdState.cCMD_READ) OR (me.intCmd=RFW_CmdState.cCMD_WRITE)) AND (SIf.Cfg.eTyp = E_Typ_RFW.RF382R) THEN
			// SIf.Alm[5].strText := 'Command for this type of RFID not possible';
			pfbAlarmCtrl^.setAlarm(CIf.Info.intCtrlId,5,UDINT_TO_DINT(pRFD_SIf^.stErr.udiErrorID),ADR(SIf.Alm),E_AlmState.RST,CIf.Job.eMe_ActivAlmClass);			
		ELSIF (me.intCmd=RFW_CmdState.cCMD_READ) THEN
			me.StateMachine.intStateNext := RFW_CmdState.cSTA_READBusy;
		ELSIF(me.intCmd=RFW_CmdState.cCMD_WRITE) THEN
			me.StateMachine.intStateNext := RFW_CmdState.cSTA_WRITEBusy;
		ELSIF(me.intCmd=RFW_CmdState.cCMD_ON) THEN
			me.StateMachine.intStateNext := RFW_CmdState.cSTA_ONBusy;			
		END_IF
	END_IF




//--------------------------------------------------------------------------------------
// Exit action
	IF (me.StateMachine.intState<>me.StateMachine.intStateNext) THEN
		;		
	END_IF
END_METHOD

METHOD PROTECTED sta_RUNbusy : BOOL
// state implemetation
//--------------------------------------------------------------------------------------
// Entry action
	IF (me.StateMachine.intState<>me.StateMachine.intStateLastCycle) THEN
		me.StateMachine.intStateLastCycle := me.StateMachine.intState;
		bolNewTag := FALSE;
		me.SubStateMachine.intState := cRFW_SUB_WaitTag;
		SIf.Cur.dwoJob := RFID_Data.cRFID_TrayID;
		
		fbSimulationTimer.IN := FALSE;
		fbSimulationTimer.PT := UDINT_TO_TIME(SIf.Par.udiReadTime_ms / 2);
		fbSimulationTimer(); // set time/reset timer
		fbSimulationTimer.IN := TRUE; // start timer
		
	END_IF


//--------------------------------------------------------------------------------------
// Cyclic action
	IF (me.StateMachine.intState=me.StateMachine.intStateLastCycle) THEN

		// Simulation
		IF (CIf.SwCfg.bolSimulation) THEN
			fbSimulationTimer(); // simulation time
			IF (fbSimulationTimer.Q) THEN
				;
			END_IF
		END_IF
		
		// Function
		
		// State Change Condition
		IF (pRFD_SIf^.stErr.bolErrorActive = TRUE) THEN  
			me.StateMachine.intStateNext :=  cSTA_ERROR;
		ELSIF(me.intCmd=cCMD_READ) THEN
			me.StateMachine.intStateNext := cSTA_READBusy;
		ELSIF(me.intCmd=cCMD_WRITE) THEN
			me.StateMachine.intStateNext := cSTA_WRITEBusy;
		ELSE
			me.StateMachine.intStateNext := cSTA_RUN;
		END_IF
	END_IF




//--------------------------------------------------------------------------------------
// Exit action
	IF (me.StateMachine.intState<>me.StateMachine.intStateNext) THEN
		;		
	END_IF
END_METHOD

METHOD PROTECTED sta_WRITE : BOOL
// state implemetation
//--------------------------------------------------------------------------------------
// Entry action
	IF (me.StateMachine.intState<>me.StateMachine.intStateLastCycle) THEN
		me.StateMachine.intStateLastCycle := me.StateMachine.intState;

	END_IF


//--------------------------------------------------------------------------------------
// Cyclic action
	IF (me.StateMachine.intState=me.StateMachine.intStateLastCycle) THEN

		// Simulation
		IF (CIf.SwCfg.bolSimulation) THEN
			;
		END_IF
		
		// State Change Condition
		IF(me.intCmd=cCMD_RUN) THEN
			me.StateMachine.intStateNext := cSTA_RUNBusy;
		ELSIF(me.intCmd=RFW_CmdState.cCMD_READ) THEN
			me.StateMachine.intStateNext := RFW_CmdState.cSTA_READBusy;
		ELSIF ((me.intCmd=RFW_CmdState.cCMD_READ) OR (me.intCmd=RFW_CmdState.cCMD_WRITE)) AND (SIf.Cfg.eTyp = E_Typ_RFW.RF382R) THEN
			// SIf.Alm[5].strText := 'Command for this type of RFID not possible';
			pfbAlarmCtrl^.setAlarm(CIf.Info.intCtrlId,5,UDINT_TO_DINT(pRFD_SIf^.stErr.udiErrorID),ADR(SIf.Alm),E_AlmState.RST,CIf.Job.eMe_ActivAlmClass);	
		ELSIF(me.intCmd=RFW_CmdState.cCMD_WRITE) THEN
			me.StateMachine.intStateNext := RFW_CmdState.cSTA_WRITEBusy;
		ELSIF(me.intCmd=RFW_CmdState.cCMD_ON) THEN
			me.StateMachine.intStateNext := RFW_CmdState.cSTA_ONBusy;			
		END_IF
	END_IF




//--------------------------------------------------------------------------------------
// Exit action
	IF (me.StateMachine.intState<>me.StateMachine.intStateNext) THEN
		;
	END_IF
END_METHOD

METHOD PROTECTED sta_WRITEBusy : BOOL
// state implemetation
//--------------------------------------------------------------------------------------
// Entry action
	IF (me.StateMachine.intState<>me.StateMachine.intStateLastCycle) THEN
		me.StateMachine.intStateLastCycle := me.StateMachine.intState;

		fbSimulationTimer.IN := FALSE;
		fbSimulationTimer.PT := UDINT_TO_TIME(SIf.Par.udiWriteTime_ms / 2);
		fbSimulationTimer(); // set time/reset timer
		fbSimulationTimer.IN := TRUE; // start timer
		
		IF SIf.Cur.dwoJob = 0 THEN
			SIf.Cur.dwoJob := RFID_Data.cRFID_AllData;
		END_IF
		
